(*
 __    __  ______  __    __  ________  __       __   ______   ________  ______   ______    ______  
/  |  /  |/      |/  \  /  |/        |/  \     /  | /      \ /        |/      | /      \  /      \ 
$$ | /$$/ $$$$$$/ $$  \ $$ |$$$$$$$$/ $$  \   /$$ |/$$$$$$  |$$$$$$$$/ $$$$$$/ /$$$$$$  |/$$$$$$  |
$$ |/$$/    $$ |  $$$  \$$ |$$ |__    $$$  \ /$$$ |$$ |__$$ |   $$ |     $$ |  $$ |  $$/ $$ \__$$/ 
$$  $$<     $$ |  $$$$  $$ |$$    |   $$$$  /$$$$ |$$    $$ |   $$ |     $$ |  $$ |      $$      \ 
$$$$$  \    $$ |  $$ $$ $$ |$$$$$/    $$ $$ $$/$$ |$$$$$$$$ |   $$ |     $$ |  $$ |   __  $$$$$$  |
$$ |$$  \  _$$ |_ $$ |$$$$ |$$ |_____ $$ |$$$/ $$ |$$ |  $$ |   $$ |    _$$ |_ $$ \__/  |/  \__$$ |
$$ | $$  |/ $$   |$$ | $$$ |$$       |$$ | $/  $$ |$$ |  $$ |   $$ |   / $$   |$$    $$/ $$    $$/ 
$$/   $$/ $$$$$$/ $$/   $$/ $$$$$$$$/ $$/      $$/ $$/   $$/    $$/    $$$$$$/  $$$$$$/   $$$$$$/  
                                                                                                   
*)

actCheckPositionDeviation();
actCheckRealSpgStatus();
actUpdateDefaults();
actClearDefaults();

startupDelayTON(PT:=T#200MS);
stateDelayTimer(PT:=T#200MS);
timeoutDelay(PT:=T#2S);

actKinematicSetpoints();
actCheckNotMoving();

GVL_INTER.TARGET_MEASUREMENT_ANGLE:= astAxes[AXIS_MEASUREMENT_ANGLE].Axis.NcToPlc.SetPos + astAxes[AXIS_MEASUREMENT_ANGLE_OFFSET].Axis.NcToPlc.SetPos + astAxes[AXIS_ROTATION_SAMPLE].Axis.NcToPlc.SetPos;


FOR i:=1 TO ARRAYSIZE_ALLVIRTUALS DO
    aVirtualAxisDefaults[i].mcSetPosition(Axis:= astAxes[aVirtualAxisDefaults[i].axisID].Axis);
    aVirtualAxisDefaults[i].mcSetPosition.Execute:= FALSE;
END_FOR

IF GVL_INTER.START_RECOVERY AND GVL_INTER.RUN_KINEMATICS AND NOT GVL_INTER.RECOVERY_IN_PROGRESS THEN
    eStateInter:= eState_INTER.startRecovery;
END_IF

IF GVL_INTER.REINITIALISE_IN_PROGRESS THEN
    GVL_INTER.REINITIALISE:= FALSE;
    GVL_INTER.START_RECOVERY:= FALSE;
END_IF
IF GVL_INTER.REINITIALISE_IN_PROGRESS AND eStateInter= eState_INTER.error THEN
    GVL_INTER.REINITIALISE_IN_PROGRESS:= FALSE;
END_IF

IF GVL_INTER.RUN_KINEMATICS AND GVL_INTER.REINITIALISE THEN
    GVL_INTER.RESET_ALL:= TRUE;
    GVL_INTER.REINITIALISE := FALSE;
    GVL_INTER.REINITIALISE_IN_PROGRESS:= TRUE;
    GVL_INTER.RUN_KINEMATICS := FALSE;
END_IF
IF GVL_INTER.FINISH_REINITIALISE AND NOT GVL_INTER.REINITIALISE_IN_PROGRESS THEN
    GVL_INTER.FINISH_REINITIALISE:= FALSE;
END_IF
IF GVL_INTER.FINISH_REINITIALISE AND GVL_INTER.REINITIALISE_IN_PROGRESS THEN
    GVL_INTER.FINISH_REINITIALISE:= FALSE;
    GVL_INTER.RUN_KINEMATICS:= TRUE;
    GVL_INTER.REINITIALISE_IN_PROGRESS:= FALSE;
    eStateInter:= eState_INTER.alignKinematics;
END_IF

IF NOT GVL_INTER.KINEMATIC_SPG_ALL_DISABLED AND NOT GVL_INTER.RUN_KINEMATICS THEN
    eStateInter:= eState_INTER.disableSPG;
END_IF


GVL_INTER.OPERATIONAL:= FALSE;  //OVERRIDE IF OPERATIONAL
IF NOT CombinedVerticalSetupComplete AND GVL_INTER.OPERATIONAL THEN
    eStateInter:= eState_INTER.init;
END_IF
checkRotationDrive(Axis:=astAxes[AXIS_ROTATION].Axis,Enable:=TRUE);

//Sometimes the rotation loads in 360degrees out of phase, we need to be able to detect and fix this.
setPosRotation(Axis:= astAxes[AXIS_ROTATION].Axis, Execute:= FALSE);

IF checkRotationDrive.Valid THEN
    IF ABS(astAxes[AXIS_ROTATION].Axis.NcToPlc.ActPos)>20 AND astAxes[AXIS_ROTATION].Axis.Status.NotMoving THEN
    astAxes[AXIS_ROTATION].stControl.bEnable:= FALSE;
    IF astAxes[AXIS_ROTATION].Axis.NcToPlc.ActPos>20 THEN
        //we need to minus 360
        setPosRotation.Position:= astAxes[AXIS_ROTATION].Axis.NcToPlc.ActPos-360;
    ELSIF astAxes[AXIS_ROTATION].Axis.NcToPlc.ActPos<20 THEN
        //we need to add 360
        setPosRotation.Position:= astAxes[AXIS_ROTATION].Axis.NcToPlc.ActPos+360;
    END_IF
    setPosRotation(Axis:= astAxes[AXIS_ROTATION].Axis, Execute:= TRUE);
ELSE
    bRotationValid:= TRUE;
END_IF
END_IF


IF NOT GVL_INTER.BRAKE_TEST_PASSED THEN
    GVL_INTER.RUN_KINEMATICS := FALSE;
END_IF    
    CASE eStateInter OF
        eState_INTER.init:       
            IF GVL_INTER.RUN_KINEMATICS AND CombinedVerticalSetupComplete AND bRotationValid THEN
                IF GVL_INTER.NC_AXIS_ERROR THEN
                    GVL_INTER.RESET_ALL := TRUE;
                    stateDelayTimer.IN:= TRUE;
                ELSIF NOT stateDelayTimer.IN THEN
                    IF NOT GVL_INTER.KINEMATIC_SPG_ALL_DISABLED THEN
                        eStateInter:=eState_INTER.disableSPG;
                    ELSE
                        IF bRealDevValid THEN
                            eStateInter:= eState_INTER.checkAlignKinematics;
                        ELSE
                            eStateInter:= eState_INTER.setPositions;
						END_IF
                        
			        END_IF
				END_IF
                //To prevent instantaneous reset and no error present
                IF stateDelayTimer.Q THEN
                    stateDelayTimer.IN:= FALSE;
				END_IF
                
			END_IF
            
                        
        eState_INTER.setPositions:
            FOR i:=1 TO ARRAYSIZE_ALLVIRTUALS DO
                aVirtualAxisDefaults[i].mcSetPosition.Position:= aVirtualAxisDefaults[i].defaultPosition ;
                aVirtualAxisDefaults[i].mcSetPosition.Execute:= TRUE;
            END_FOR            
            writeDefault.START:=TRUE;            
            stateDelayTimer.IN:= TRUE;
            IF(stateDelayTimer.Q) THEN
                eStateInter := eState_INTER.checkSetPositions;
                stateDelayTimer.IN:= FALSE;
			END_IF
            
        
        eState_INTER.checkSetPositions:
            IF bDefaultDevValid THEN
                retryCounter:= 0;
                IF bRealDevValid THEN
                    eStateInter:= eState_INTER.enableSPG;
                ELSE
                    eStateInter:= eState_INTER.alignKinematics;
			    END_IF
            ELSE
                IF retryCounter >3 THEN
                    retryCounter:= 0;
                    eStateInter:= eState_INTER.error;
                    GVL_INTER.LOGIC_STATE_ERROR:= eState_INTER.checkSetPositions;
                    GVL_INTER.LOGIC_ERROR:= TRUE;
                ELSE
                    retryCounter:= retryCounter+1;
                    eStateInter:= eState_INTER.setPositions;
				END_IF                
			END_IF               


        eState_INTER.alignKinematics:
            startupDelayTON.IN:= TRUE;
            IF startupDelayTON.Q THEN
                startupDelayTON.IN:= FALSE;
                AbsoluteMove(axisID:= AXIS_HORIZONTAL_TRANSLATION, fPosition:= GVL_INTER.SETPOS_HORIZONTAL);
                AbsoluteMove(axisID:= AXIS_COMBINED_VERTICAL, fPosition:= GVL_INTER.SETPOS_COMBINED_VERTICAL);
                AbsoluteMove(axisID:= AXIS_ROTATION, fPosition:= GVL_INTER.SETPOS_ROTATION);               
                stateDelayTimer.IN:= TRUE;
			END_IF
            IF stateDelayTimer.Q THEN
                eStateInter:= eState_INTER.checkAlignKinematics;
                stateDelayTimer.IN:= FALSE;
			END_IF
            IF NOT (startupDelayTON.IN OR stateDelayTimer.IN) THEN
                GVL_INTER.LOGIC_STATE_ERROR:= eState_INTER.alignKinematics;
                GVL_INTER.LOGIC_ERROR:= TRUE;
                eStateInter:= eState_INTER.error;
			END_IF
            

        eState_INTER.checkAlignKinematics:
            IF GVL_INTER.REAL_AXES_NOT_MOVING THEN   
                timeoutDelay.IN:= TRUE;            
                IF bRealDevValid THEN
                    timeoutDelay.IN:= FALSE;
                    eStateInter:= eState_INTER.enableSPG;
		        END_IF
                IF GVL_INTER.LIMIT_HIT THEN
                    timeoutDelay.IN:= FALSE;
                    GVL_INTER.LOGIC_STATE_ERROR:= eState_INTER.checkAlignKinematics;
                    GVL_INTER.LOGIC_ERROR:= TRUE;
                    eStateInter:= eState_INTER.error;
				END_IF
                IF timeoutDelay.Q THEN
                    timeoutDelay.IN:= FALSE;
                    GVL_INTER.LOGIC_STATE_ERROR:= eState_INTER.checkAlignKinematics;
                    GVL_INTER.LOGIC_ERROR:= TRUE;
                    eStateInter:= eState_INTER.error;
				END_IF
		    END_IF
                
            
        eState_INTER.enableSPG:
            axisSpg_Vertical.spgEnable.Execute:= TRUE;
            axisSpg_Horizontal.spgEnable.Execute:= TRUE;
            axisSpg_Rot.spgEnable.Execute:= TRUE;
            stateDelayTimer.IN:= TRUE;
            IF stateDelayTimer.Q THEN
                stateDelayTimer.IN:= FALSE;
                eStateInter:= eState_INTER.checkEnableSPG;
			END_IF
            
           
        eState_INTER.checkEnableSPG:
            IF GVL_INTER.KINEMATIC_SPG_ALL_ENABLED THEN
                retryCounter:= 0;
                eStateInter :=eState_INTER.operation;
            ELSE
                IF retryCounter >3 THEN
                    retryCounter:= 0;
                    eStateInter:= eState_INTER.error;
                    GVL_INTER.LOGIC_STATE_ERROR:= eState_INTER.checkEnableSPG;
                    GVL_INTER.LOGIC_ERROR:= TRUE;
                ELSE
                    retryCounter:= retryCounter+1;
                    eStateInter:= eState_INTER.enableSPG;
		        END_IF 
			END_IF
            
        
        eState_INTER.operation:
            GVL_INTER.RECOVERY_IN_PROGRESS:= FALSE;
            bKinematicsOperational:= TRUE;
            IF NOT GVL_INTER.KINEMATIC_SPG_ALL_ENABLED THEN
                eStateInter:= eState_INTER.error;
			END_IF
            IF NOT GVL_INTER.NC_AXIS_ERROR THEN
                GVL_INTER.OPERATIONAL:= TRUE;
            END_IF
            
        eState_INTER.disableSPG:
            axisSpg_Vertical.spgDisable.Execute:= TRUE;
            axisSpg_Horizontal.spgDisable.Execute:= TRUE;
            axisSpg_Rot.spgDisable.Execute:= TRUE;
            stateDelayTimer.IN:= TRUE;
            IF stateDelayTimer.Q THEN
                stateDelayTimer.IN:= FALSE;
                eStateInter:= eState_INTER.checkDisableSPG;
			END_IF
            
        eState_INTER.checkDisableSPG:
            IF GVL_INTER.KINEMATIC_SPG_ALL_DISABLED THEN
                retryCounter:= 0;
                IF GVL_INTER.RECOVERY_IN_PROGRESS THEN
                    eStateInter:= eState_INTER.recoveryDefaultPosition;
                ELSE
                    eStateInter:= eState_INTER.init;
				END_IF
            ELSE
                IF retryCounter >3 THEN
                    retryCounter:= 0;
                    eStateInter:= eState_INTER.error;
                    GVL_INTER.LOGIC_STATE_ERROR:= eState_INTER.checkDisableSPG;
                    GVL_INTER.LOGIC_ERROR:= TRUE;
                ELSE
                    retryCounter:= retryCounter+1;
                    eStateInter:= eState_INTER.disableSPG;
		        END_IF 
			END_IF
            
        eState_INTER.startRecovery:
            GVL_INTER.RECOVERY_IN_PROGRESS := TRUE;
            eStateInter:= eState_INTER.disableSPG;
        
        eState_INTER.recoveryDefaultPosition:
            IF GVL_INTER.NC_AXIS_ERROR THEN
                GVL_INTER.RESET_ALL := TRUE;
            ELSE
                FOR i:=1 TO ARRAYSIZE_ALLVIRTUALS DO
                    aVirtualAxisDefaults[i].mcSetPosition.Position:= aVirtualAxisDefaults[i].defaultPosition;
                    aVirtualAxisDefaults[i].mcSetPosition.Execute:= TRUE;
                    aVirtualAxisDefaults[i].mcSetPosition.Options.ClearPositionLag:= TRUE;
                END_FOR
                
                stateDelayTimer.IN:= TRUE;
                IF stateDelayTimer.Q THEN
                    stateDelayTimer.IN:= FALSE;
                    eStateInter:= eState_INTER.waitForRecovery;
			    END_IF
			END_IF
            
          
        eState_INTER.waitForRecovery:
            IF GVL_INTER.VIRTUAL_AXES_NOT_MOVING THEN                
                timeoutDelay.IN:= TRUE;            
                IF bRecoveryDevValid THEN
                    timeoutDelay.IN:= FALSE;
                    GVL_INTER.START_RECOVERY:= FALSE;                    
                    eStateInter:= eState_INTER.init;                                
			    END_IF
                
                IF timeoutDelay.Q THEN
                    timeoutDelay.IN:= FALSE;
                    GVL_INTER.LOGIC_STATE_ERROR:= eState_INTER.waitForRecovery;
                    GVL_INTER.LOGIC_ERROR:= TRUE;
                    GVL_INTER.START_RECOVERY:= FALSE;
                    GVL_INTER.RECOVERY_IN_PROGRESS:= FALSE;
                    eStateInter:= eState_INTER.error;
				END_IF           
			END_IF
            
            
        eState_INTER.error:
            GVL_INTER.RECOVERY_IN_PROGRESS:= FALSE;
            IF GVL_INTER.RESET_REQUESTED THEN
                eStateInter:= eState_INTER.safetyError;
			END_IF
            IF GVL_INTER.ACKNOWLEDGE_LOGIC_ERROR THEN
                GVL_INTER.ACKNOWLEDGE_LOGIC_ERROR := FALSE;
                GVL_INTER.LOGIC_STATE_ERROR:= eState_INTER.none;
                GVL_INTER.LOGIC_ERROR:= FALSE;
                GVL_INTER.RESET_ALL:= TRUE;
			END_IF
            IF GVL_Safety.LocalMode AND GVL_Safety.LocalMode_Disabled THEN
                eStateInter:= eState_INTER.localModeDisabled;
			END_IF
            IF NOT GVL_INTER.NC_AXIS_ERROR  AND NOT GVL_INTER.LOGIC_ERROR THEN
                eStateInter:= eState_INTER.init;
			END_IF
            
        eState_INTER.localModeDisabled:
            IF NOT GVL_INTER.NC_AXIS_ERROR  AND NOT GVL_INTER.LOGIC_ERROR THEN
                eStateInter:= eState_INTER.init;
			END_IF
            
        eState_INTER.safetyError:
            GVL_INTER.RUN_KINEMATICS:= FALSE;
            IF GVL_INTER.ACKNOWLEDGE_LOGIC_ERROR THEN
                GVL_INTER.ACKNOWLEDGE_LOGIC_ERROR := FALSE;
                GVL_INTER.LOGIC_STATE_ERROR:= eState_INTER.none;
                GVL_INTER.LOGIC_ERROR:= FALSE;
                GVL_INTER.RESET_ALL:= TRUE;
			END_IF
            IF NOT GVL_INTER.NC_AXIS_ERROR  AND NOT GVL_INTER.LOGIC_ERROR THEN
                eStateInter:= eState_INTER.init;
			END_IF
            
	END_CASE
    
    IF GVL_INTER.REINITIALISE_IN_PROGRESS OR GVL_INTER.OPERATIONAL THEN   
        FOR i:=1 TO ARRAYSIZE_ALLVIRTUALS DO
            astAxes[aVirtualAxisDefaults[i].axisID].stControl.bEnable:=TRUE;
            astAxes[aVirtualAxisDefaults[i].axisID].stInputs.bLimitBwd:=TRUE;
            astAxes[aVirtualAxisDefaults[i].axisID].stInputs.bLimitFwd:=TRUE;
		END_FOR
    ELSE
        FOR i:=1 TO ARRAYSIZE_ALLVIRTUALS DO
            astAxes[aVirtualAxisDefaults[i].axisID].stControl.bEnable:=FALSE;
            astAxes[aVirtualAxisDefaults[i].axisID].stInputs.bLimitBwd:=FALSE;
            astAxes[aVirtualAxisDefaults[i].axisID].stInputs.bLimitFwd:=FALSE;
		END_FOR
	END_IF

 
//Call set position functions on virtual axes
FOR i:=1 TO ARRAYSIZE_ALLVIRTUALS DO
    aVirtualAxisDefaults[i].mcSetPosition(Axis:=astAxes[aVirtualAxisDefaults[i].axisID].Axis);
    aVirtualAxisDefaults[i].mcSetPosition.Execute:= FALSE;
END_FOR   

GVL_INTER.LOGIC_STATE_STR := TO_STRING(GVL_INTER.LOGIC_STATE);
GVL_INTER.LOGIC_STATE_ERROR_STR := TO_STRING(GVL_INTER.LOGIC_STATE_ERROR);


MC_ExtSetPointGenFeed(Axis:= astAxes[AXIS_COMBINED_VERTICAL].Axis, 
        Position:= axisSpg_Vertical.position,
        Velocity:= axisSpg_Vertical.velocity,
        Direction:= axisSpg_Vertical.direction, Acceleration:= 0);
MC_ExtSetPointGenFeed(Axis:= astAxes[AXIS_HORIZONTAL_TRANSLATION].Axis, 
        Position:= axisSpg_Horizontal.position,
        Velocity:= axisSpg_Horizontal.velocity,
        Direction:= axisSpg_Horizontal.direction, Acceleration:= 0);
MC_ExtSetPointGenFeed(Axis:= astAxes[AXIS_ROTATION].Axis, 
        Position:= axisSpg_Rot.position,
        Velocity:= axisSpg_Rot.velocity,
        Direction:= axisSpg_Rot.direction, Acceleration:= 0);

axisSpg_Vertical.spgEnable(Axis:=astAxes[axisSpg_Vertical.axisID].Axis);
axisSpg_Vertical.spgDisable(Axis:=astAxes[axisSpg_Vertical.axisID].Axis);
axisSpg_Horizontal.spgEnable(Axis:=astAxes[axisSpg_Horizontal.axisID].Axis);
axisSpg_Horizontal.spgDisable(Axis:=astAxes[axisSpg_Horizontal.axisID].Axis);
axisSpg_Rot.spgEnable(Axis:=astAxes[axisSpg_Rot.axisID].Axis);
axisSpg_Rot.spgDisable(Axis:=astAxes[axisSpg_Rot.axisID].Axis);

axisSpg_Vertical.spgEnable.Execute:= FALSE;
axisSpg_Vertical.spgDisable.Execute:= FALSE;
axisSpg_Horizontal.spgEnable.Execute:= FALSE;
axisSpg_Horizontal.spgDisable.Execute:= FALSE;
axisSpg_Rot.spgEnable.Execute:= FALSE;
axisSpg_Rot.spgDisable.Execute:= FALSE;

GVL_INTER.LOGIC_STATE:= eStateInter;

IF ABS( astAxes[AXIS_VERTICAL_TRANSLATION_Y1].stStatus.fActPosition-astAxes[AXIS_VERTICAL_TRANSLATION_Y2].stStatus.fActPosition)>3 THEN
    astAxes[AXIS_COMBINED_VERTICAL].stControl.bEnable:= FALSE;
END_IF

METHOD AbsoluteMove : BOOL
VAR_INPUT
    axisID : UINT;
    fPosition : LREAL;
    
END_VAR
astAxes[axisID].stControl.eCommand:= E_MotionFunctions.eMoveAbsolute;
astAxes[axisID].stControl.fPosition:= fPosition;
astAxes[axisID].stControl.bExecute:= TRUE;
END_METHOD

ACTION actCheckNotMoving:
GVL_INTER.REAL_AXES_NOT_MOVING:= astAxes[AXIS_HORIZONTAL_TRANSLATION].Axis.Status.NotMoving AND astAxes[AXIS_COMBINED_VERTICAL].Axis.Status.NotMoving AND astAxes[AXIS_ROTATION].Axis.Status.NotMoving;

GVL_INTER.VIRTUAL_AXES_NOT_MOVING:= 
    astAxes[AXIS_DOFF_ANGLED].Axis.Status.NotMoving AND
    astAxes[AXIS_DOFF_PARALLEL].Axis.Status.NotMoving AND
    astAxes[AXIS_DTANK_LENGTH].Axis.Status.NotMoving AND
    astAxes[AXIS_DTANK_PIVOT_TO_WINDOW].Axis.Status.NotMoving AND
    astAxes[AXIS_DRAD].Axis.Status.NotMoving AND
    astAxes[AXIS_MEASUREMENT_ANGLE].Axis.Status.NotMoving AND
    astAxes[AXIS_MEASUREMENT_ANGLE_OFFSET].Axis.Status.NotMoving AND
    astAxes[AXIS_ROTATION_CALIBRATION].Axis.Status.NotMoving AND
    astAxes[AXIS_ROTATION_SAMPLE].Axis.Status.NotMoving AND
    astAxes[AXIS_COMBINED_VERTICAL_CALIBRATION].Axis.Status.NotMoving AND
    astAxes[AXIS_COMBINED_VERTICAL_SAMPLE].Axis.Status.NotMoving AND
    astAxes[AXIS_HORIZONTAL_CALIBRATION].Axis.Status.NotMoving AND
    astAxes[AXIS_HORIZONTAL_SAMPLE].Axis.Status.NotMoving;
END_ACTION

ACTION actCheckPositionDeviation:
posDevHorizontal:=    astAxes[AXIS_HORIZONTAL_TRANSLATION].stStatus.fActPosition - GVL_INTER.SETPOS_HORIZONTAL;
posDevVertical:=    astAxes[AXIS_COMBINED_VERTICAL].stStatus.fActPosition - GVL_INTER.SETPOS_COMBINED_VERTICAL;
posDevRot:=    astAxes[AXIS_ROTATION].stStatus.fActPosition - GVL_INTER.SETPOS_ROTATION;

bRealDevValid := ABS(posDevHorizontal)<DEVIATION_THRESHOLD AND ABS(posDevVertical)<DEVIATION_THRESHOLD AND ABS(posDevRot)<DEVIATION_THRESHOLD;

(*
//Check position deviations of "default" axes
bDefaultDevValid:= TRUE; //we will AND it with the deviations in the loop
FOR i := 1 TO ARRAYSIZE_VIRTUALCAL DO
    bDefaultDevValid:= bDefaultDevValid AND (ABS(astAxes[IDs_VirtualWithCalibrationAxes[i]].stStatus.fActPosition - calibrationValuesArray[i])<DEVIATION_THRESHOLD);
END_FOR


//Check position deviations of remaining virtual axes
bRecoveryDevValid:= bDefaultDevValid; //Use default dev as starting point before iterator
FOR i := 1 TO ARRAYSIZE_VIRTUAL DO
    bRecoveryDevValid:= bRecoveryDevValid AND (ABS(astAxes[IDs_VirtualNoCalibrationAxes[i]].stStatus.fActPosition)<DEVIATION_THRESHOLD);
END_FOR
*)

////
////
////
//THIS IS NEW LOGIC THAT OVERRIDES WHAT'S CURRENTLY HAPPENING, BE CAREFUL
bRecoveryDevValid:= TRUE;
FOR i:=1 TO ARRAYSIZE_ALLVIRTUALS DO
    aVirtualAxisDefaults[i].deviation:= ABS(astAxes[aVirtualAxisDefaults[i].axisID].Axis.NcToPlc.ActPos - aVirtualAxisDefaults[i].defaultPosition);
    bRecoveryDevValid:= bRecoveryDevValid AND (aVirtualAxisDefaults[i].deviation<DEVIATION_THRESHOLD);
END_FOR

bDefaultDevValid := bRecoveryDevValid;

bVirtualsMoving:= FALSE;
FOR i := 1 TO ARRAYSIZE_ALLVIRTUALS DO
    bVirtualsMoving:= bVirtualsMoving OR astAxes[aVirtualAxisDefaults[i].axisID].Axis.Status.Moving;
END_FOR
/////
/////
/////
    
    
//bVirtualsMoving:= FALSE;
//Looking for any virtual axis moving IDs_VirtualNoCalibrationAxes
//FOR i := 1 TO ARRAYSIZE_VIRTUALCAL DO
//    bVirtualsMoving:= bVirtualsMoving OR astAxes[IDs_VirtualWithCalibrationAxes[i]].Axis.Status.Moving;
//END_FOR
//FOR i := 1 TO ARRAYSIZE_VIRTUAL DO
//    bVirtualsMoving:= bVirtualsMoving OR astAxes[IDs_VirtualNoCalibrationAxes[i]].Axis.Status.Moving;
//END_FOR
END_ACTION

ACTION actCheckRealSpgStatus:
GVL_INTER.KINEMATIC_SPG_ALL_ENABLED:= astAxes[AXIS_HORIZONTAL_TRANSLATION].Axis.Status.ExtSetPointGenEnabled AND astAxes[AXIS_COMBINED_VERTICAL].Axis.Status.ExtSetPointGenEnabled AND astAxes[AXIS_ROTATION].Axis.Status.ExtSetPointGenEnabled;
GVL_INTER.KINEMATIC_SPG_ALL_DISABLED:= NOT (astAxes[AXIS_HORIZONTAL_TRANSLATION].Axis.Status.ExtSetPointGenEnabled) AND NOT (astAxes[AXIS_COMBINED_VERTICAL].Axis.Status.ExtSetPointGenEnabled) AND NOT (astAxes[AXIS_ROTATION].Axis.Status.ExtSetPointGenEnabled);
END_ACTION

ACTION actClearDefaults:
IF GVL_INTER.CLEAR_ALL_DEFAULTS THEN
    IF NOT bVirtualsMoving THEN
        GVL_INTER.CLEAR_ALL_DEFAULTS:= FALSE;   
        aVirtualAxisDefaults[1].defaultPosition:= 3000;
        aVirtualAxisDefaults[2].defaultPosition:= 2289.15;
        aVirtualAxisDefaults[3].defaultPosition:= 1648.66;
        aVirtualAxisDefaults[4].defaultPosition:= 0;
        aVirtualAxisDefaults[5].defaultPosition:= 0;
        aVirtualAxisDefaults[6].defaultPosition:= 0;
        aVirtualAxisDefaults[7].defaultPosition:= 0;
        aVirtualAxisDefaults[8].defaultPosition:= 0;
        aVirtualAxisDefaults[9].defaultPosition:= 0;
        aVirtualAxisDefaults[10].defaultPosition:= 0;
        aVirtualAxisDefaults[11].defaultPosition:= 0;
        aVirtualAxisDefaults[12].defaultPosition:= 0;
        aVirtualAxisDefaults[13].defaultPosition:= 0;
	END_IF
END_IF
END_ACTION

ACTION actKinematicSetpoints:
(*GVL_INTER.SETPOS_HORIZONTAL:= astAxes[AXIS_HORIZONTAL_VIRTUAL].Axis.NcToPlc.ActPos + astAxes[AXIS_HORIZONTAL_CALIBRATION].Axis.NcToPlc.ActPos + astAxes[AXIS_HORIZONTAL_SAMPLE].Axis.NcToPlc.ActPos;
GVL_INTER.SETVELO_HORIZONTAL:=astAxes[AXIS_HORIZONTAL_VIRTUAL].Axis.NcToPlc.ActVelo + astAxes[AXIS_HORIZONTAL_CALIBRATION].Axis.NcToPlc.ActVelo + astAxes[AXIS_HORIZONTAL_SAMPLE].Axis.NcToPlc.ActVelo;
GVL_INTER.SETPOS_COMBINED_VERTICAL:= astAxes[AXIS_COMBINED_VERTICAL_VIRTUAL].Axis.NcToPlc.ActPos + astAxes[AXIS_COMBINED_VERTICAL_CALIBRATION].Axis.NcToPlc.ActPos + astAxes[AXIS_COMBINED_VERTICAL_SAMPLE].Axis.NcToPlc.ActPos;
GVL_INTER.SETVELO_COMBINED_VERTICAL:= astAxes[AXIS_COMBINED_VERTICAL_VIRTUAL].Axis.NcToPlc.ActVelo + astAxes[AXIS_COMBINED_VERTICAL_CALIBRATION].Axis.NcToPlc.ActVelo + astAxes[AXIS_COMBINED_VERTICAL_SAMPLE].Axis.NcToPlc.ActVelo;
GVL_INTER.SETPOS_ROTATION:= astAxes[AXIS_ROTATION_VIRTUAL].Axis.NcToPlc.ActPos + astAxes[AXIS_ROTATION_CALIBRATION].Axis.NcToPlc.ActPos + astAxes[AXIS_ROTATION_SAMPLE].Axis.NcToPlc.ActPos;
GVL_INTER.SETVELO_ROTATION:= astAxes[AXIS_ROTATION_VIRTUAL].Axis.NcToPlc.ActVelo + astAxes[AXIS_ROTATION_CALIBRATION].Axis.NcToPlc.ActVelo + astAxes[AXIS_ROTATION_SAMPLE].Axis.NcToPlc.ActVelo;

//Horizontal direction
IF GVL_INTER.SETVELO_HORIZONTAL >0 THEN
    GVL_INTER.SETDIR_HORIZONTAL := 1;
ELSIF GVL_INTER.SETVELO_HORIZONTAL<0 THEN
    GVL_INTER.SETDIR_HORIZONTAL := -1;
ELSE
    GVL_INTER.SETDIR_HORIZONTAL := 0;
END_IF

//Vertical Direction
IF GVL_INTER.SETVELO_COMBINED_VERTICAL>0 THEN
    GVL_INTER.SETDIR_COMBINED_VERTICAL := 1;
ELSIF GVL_INTER.SETVELO_COMBINED_VERTICAL<0 THEN
    GVL_INTER.SETDIR_COMBINED_VERTICAL := -1;
ELSE
    GVL_INTER.SETDIR_COMBINED_VERTICAL := 0;
END_IF

//Rotation direction
IF GVL_INTER.SETVELO_ROTATION>0 THEN
    GVL_INTER.SETDIR_ROTATION := 1;
ELSIF GVL_INTER.SETVELO_ROTATION<0 THEN
    GVL_INTER.SETDIR_ROTATION := -1;
ELSE
    GVL_INTER.SETDIR_ROTATION := 0;
END_IF
*)

//NEW LOGIC
axisSpg_Vertical.position:= astAxes[AXIS_COMBINED_VERTICAL_VIRTUAL].Axis.NcToPlc.ActPos + astAxes[AXIS_COMBINED_VERTICAL_CALIBRATION].Axis.NcToPlc.ActPos + astAxes[AXIS_COMBINED_VERTICAL_SAMPLE].Axis.NcToPlc.ActPos;
axisSpg_Horizontal.position:= astAxes[AXIS_HORIZONTAL_VIRTUAL].Axis.NcToPlc.ActPos + astAxes[AXIS_HORIZONTAL_CALIBRATION].Axis.NcToPlc.ActPos + astAxes[AXIS_HORIZONTAL_SAMPLE].Axis.NcToPlc.ActPos;
//axisSpg_Rot.position:= astAxes[AXIS_ROTATION_VIRTUAL].Axis.NcToPlc.ActPos + astAxes[AXIS_ROTATION_CALIBRATION].Axis.NcToPlc.ActPos + astAxes[AXIS_ROTATION_SAMPLE].Axis.NcToPlc.ActPos;

axisSpg_Rot.position:= astAxes[AXIS_ROTATION_VIRTUAL].Axis.NcToPlc.ActPos + astAxes[AXIS_ROTATION_CALIBRATION].Axis.NcToPlc.ActPos;

axisSpg_Vertical.velocity:= astAxes[AXIS_COMBINED_VERTICAL_VIRTUAL].Axis.NcToPlc.ActVelo + astAxes[AXIS_COMBINED_VERTICAL_CALIBRATION].Axis.NcToPlc.ActVelo + astAxes[AXIS_COMBINED_VERTICAL_SAMPLE].Axis.NcToPlc.ActVelo;
axisSpg_Horizontal.velocity:=astAxes[AXIS_HORIZONTAL_VIRTUAL].Axis.NcToPlc.ActVelo + astAxes[AXIS_HORIZONTAL_CALIBRATION].Axis.NcToPlc.ActVelo + astAxes[AXIS_HORIZONTAL_SAMPLE].Axis.NcToPlc.ActVelo;
//axisSpg_Rot.velocity:= astAxes[AXIS_ROTATION_VIRTUAL].Axis.NcToPlc.ActVelo + astAxes[AXIS_ROTATION_CALIBRATION].Axis.NcToPlc.ActVelo + astAxes[AXIS_ROTATION_SAMPLE].Axis.NcToPlc.ActVelo;
axisSpg_Rot.velocity:= astAxes[AXIS_ROTATION_VIRTUAL].Axis.NcToPlc.ActVelo + astAxes[AXIS_ROTATION_CALIBRATION].Axis.NcToPlc.ActVelo;

//Horizontal direction
IF axisSpg_Horizontal.velocity >0 THEN
    axisSpg_Horizontal.direction := 1;
ELSIF axisSpg_Horizontal.velocity<0 THEN
    axisSpg_Horizontal.direction := -1;
ELSE
    axisSpg_Horizontal.direction := 0;
END_IF

//Vertical direction
IF axisSpg_Vertical.velocity >0 THEN
    axisSpg_Vertical.direction := 1;
ELSIF axisSpg_Vertical.velocity<0 THEN
    axisSpg_Vertical.direction := -1;
ELSE
    axisSpg_Vertical.direction := 0;
END_IF

//Rotation direction
IF axisSpg_Rot.velocity >0 THEN
    axisSpg_Rot.direction := 1;
ELSIF axisSpg_Rot.velocity<0 THEN
    axisSpg_Rot.direction := -1;
ELSE
    axisSpg_Rot.direction := 0;
END_IF


//Transfer values over to GVL_INTER
GVL_INTER.SETPOS_HORIZONTAL:=axisSpg_Horizontal.position;
GVL_INTER.SETVELO_HORIZONTAL:=axisSpg_Horizontal.velocity;
GVL_INTER.SETDIR_HORIZONTAL:= axisSpg_Horizontal.direction;

GVL_INTER.SETPOS_COMBINED_VERTICAL:= axisSpg_Vertical.position;
GVL_INTER.SETVELO_COMBINED_VERTICAL:= axisSpg_Vertical.velocity;
GVL_INTER.SETDIR_COMBINED_VERTICAL:= axisSpg_Vertical.direction;

GVL_INTER.SETPOS_ROTATION:= axisSpg_Rot.position;
GVL_INTER.SETVELO_ROTATION:= axisSpg_Rot.velocity;
GVL_INTER.SETDIR_ROTATION:= axisSpg_Rot.direction;
END_ACTION

ACTION actSafeSpeedSwitching:
IF GVL_Safety.UnoccupiedMode THEN
    //HIGH SPEED
    //MEASUREMENT AXIS valid at 0.65 degs/s  
    //Verts max at 27.5
    //Rot at 0.65
    //Hor at 1.3
    //
    FOR i:=1 TO ARRAYSIZE_ALLVIRTUALS DO
        astAxes[aVirtualAxisDefaults[i].axisID].stConfig.fOverride := 100;
        GVL_INTER.SPEED_LIMITING:= FALSE;
	END_FOR
ELSE
    //LOW SPEED
    FOR i:=1 TO ARRAYSIZE_ALLVIRTUALS DO
        astAxes[aVirtualAxisDefaults[i].axisID].stConfig.fOverride := LOCALMODE_SPEED_OVERRIDE * LOCALMODE_SPEED_OVERRIDE_MODIFIER;
        GVL_INTER.SPEED_LIMITING:= TRUE;
	END_FOR
END_IF



(*
//Check speeds not too high
IF NOT GVL_INTER.SPEED_LIMITING AND (ABS(axisSpg_Vertical.velocity)>VERTICAL_SPEED_LIMIT OR ABS(axisSpg_Horizontal.velocity)>HORIZONTAL_SPEED_LIMIT OR ABS(axisSpg_Rot.velocity)>ROTATION_SPEED_LIMIT) THEN
    IF axisSpg_Vertical.velocity>0 THEN
        axisSpg_Vertical.velocity:= VERTICAL_SPEED_LIMIT;
    ELSE
        axisSpg_Vertical.velocity:= -VERTICAL_SPEED_LIMIT;
    END_IF    
    
    IF axisSpg_Horizontal.velocity>0 THEN
        axisSpg_Horizontal.velocity:= HORIZONTAL_SPEED_LIMIT;
    ELSE
        axisSpg_Horizontal.velocity:= -HORIZONTAL_SPEED_LIMIT;
    END_IF 
    
     IF axisSpg_Rot.velocity>0 THEN
        axisSpg_Rot.velocity:= ROTATION_SPEED_LIMIT;
    ELSE
        axisSpg_Rot.velocity:= -ROTATION_SPEED_LIMIT;
    END_IF 

    FOR i:=1 TO ARRAYSIZE_ALLVIRTUALS DO
        astAxes[aVirtualAxisDefaults[i].axisID].stConfig.fOverride := 20;
        GVL_INTER.SPEED_LIMITING:= TRUE;
	END_FOR
END_IF
//We have stopped moving so can stop speed limiting
IF GVL_INTER.VIRTUAL_AXES_NOT_MOVING AND GVL_INTER.SPEED_LIMITING THEN
    FOR i:=1 TO ARRAYSIZE_ALLVIRTUALS DO
        astAxes[aVirtualAxisDefaults[i].axisID].stConfig.fOverride := 100;
        GVL_INTER.SPEED_LIMITING:= FALSE;
	END_FOR
END_IF
*)
END_ACTION

ACTION actSyncVertStateMachine:
CombinedVerticalSetupComplete := FALSE;
vertTon(PT:=T#100MS);
vertDelay(PT:=T#100MS);
CASE eStateVertical OF
        eState_Vertical.init:
            IF NOT astAxes[AXIS_VERTICAL_TRANSLATION_Y1].Axis.STatus.Error OR NOT astAxes[AXIS_VERTICAL_TRANSLATION_Y2].Axis.Status.Error THEN
                IF NOT GVL_INTER.DECOUPLE_VERTICAL_AXES THEN
                    eStateVertical := eState_Vertical.checkPosition;
                END_IF
			END_IF
            
        eState_Vertical.checkPosition:
            vertDelay.IN:= TRUE;
            IF ABS(astAxes[AXIS_VERTICAL_TRANSLATION_Y1].stStatus.fActPosition - astAxes[AXIS_VERTICAL_TRANSLATION_Y2].stStatus.fActPosition)>0.02 THEN
                AbsoluteMove(axisID:=AXIS_VERTICAL_TRANSLATION_Y2,fPosition:= astAxes[AXIS_VERTICAL_TRANSLATION_Y1].stStatus.fActPosition);
			    bVertCorrectionInProgress:= TRUE;
            END_IF
            IF vertDelay.Q AND astAxes[AXIS_VERTICAL_TRANSLATION_Y2].Axis.Status.NotMoving THEN
                bVertCorrectionInProgress:= FALSE;
			END_IF
            IF NOT bVertCorrectionInProgress THEN
                vertDelay.IN:= FALSE;
                eStateVertical := eState_Vertical.setPosition; //should be setPosition state
			END_IF
            
            //Assume Z1 and Z2 calibrated to be at same position
            //IF ABS(fVerticalSimulatedDeviation)> fVerticalSimulatedDeviationAllowed THEN
            //ELSE
                //eStateVertical := eState_Vertical.enableSpg;
			//END_IF
            
        eState_Vertical.setPosition:
            combinedVerticalSetPos.Position:= astAxes[AXIS_VERTICAL_TRANSLATION_Y1].stStatus.fActPosition;
            combinedVerticalSetPos.Execute:= TRUE;
            //eStateVertical := eState_Vertical.checkPosition;
            vertTon.In := TRUE;
            IF vertTon.Q THEN
                eStateVertical := eState_Vertical.enableSpg;
                vertTon.IN:= FALSE;
			END_IF
            
            
        eState_Vertical.enableSpg:
        
            IF astAxes[AXIS_COMBINED_VERTICAL].stInputs.bLimitBwd AND astAxes[AXIS_COMBINED_VERTICAL].stInputs.bLimitFwd THEN
                verticalZ1SpgEnable.Execute := TRUE;
                verticalZ2SpgEnable.Execute := TRUE;
                eStateVertical := eState_Vertical.confirmEnableSpg;
            ELSE
                tempZ1Power(Axis:= astAxes[AXIS_VERTICAL_TRANSLATION_Y1].Axis, Enable:= TRUE, Enable_Negative:=TRUE, Enable_Positive:=TRUE);
			    tempZ2Power(Axis:= astAxes[AXIS_VERTICAL_TRANSLATION_Y2].Axis, Enable:= TRUE, Enable_Negative:=TRUE, Enable_Positive:=TRUE);
                verticalZ1SpgEnable.Execute := TRUE;
                verticalZ2SpgEnable.Execute := TRUE;
                eStateVertical := eState_Vertical.confirmEnableSpg;
            END_IF
            
        
        eState_Vertical.confirmEnableSpg:
            confirmSpgTimeout.IN:= TRUE;
            //Timeout check
            IF confirmSpgTimeout.Q THEN
                confirmSpgTimeout.IN:= FALSE;
                eStateVertical := eState_Vertical.init;
			END_IF
            IF VerticalAxesSpgEnabled THEN
                eStateVertical := eState_Vertical.operation;
			END_IF
        
        eState_Vertical.operation:
            //DO NOTHING
            CombinedVerticalSetupComplete := TRUE;
            IF NOT VerticalAxesSpgEnabled THEN
                eStateVertical:= eState_Vertical.init;
			END_IF
            IF astAxes[AXIS_VERTICAL_TRANSLATION_Y1].Axis.STatus.Error OR astAxes[AXIS_VERTICAL_TRANSLATION_Y2].Axis.Status.Error THEN
                eStateVertical:= eState_Vertical.init;
			END_IF
            IF GVL_INTER.DECOUPLE_VERTICAL_AXES THEN
                eStateVertical := eState_Vertical.disableSpg;
			END_IF
            (*IF astAxes[AXIS_COMBINED_VERTICAL].Axis.Status.NotMoving THEN
                IF ABS(astAxes[AXIS_COMBINED_VERTICAL].stStatus.fActPosition-astAxes[AXIS_VERTICAL_TRANSLATION_Y1].stStatus.fActPosition)>0.02 THEN
                    combinedVerticalSetPos.Position:= astAxes[AXIS_VERTICAL_TRANSLATION_Y1].stStatus.fActPosition;
                    combinedVerticalSetPos.Execute:= TRUE;
				END_IF
			END_IF*)
            
        eState_Vertical.disableSpg:
            verticalZ1SpgDisable.Execute:= TRUE;
            verticalZ2SpgDisable.Execute:= TRUE;
            eStateVertical := eState_Vertical.confirmDisableSpg;
            
        eState_Vertical.confirmDisableSpg:
            IF NOT astAxes[AXIS_VERTICAL_TRANSLATION_Y1].Axis.Status.ExtSetPointGenEnabled AND NOT astAxes[AXIS_VERTICAL_TRANSLATION_Y2].Axis.Status.ExtSetPointGenEnabled THEN
                eStateVertical := eState_Vertical.init;
            ELSE
                eStateVertical := eState_Vertical.disableSpg;
			END_IF
            
	END_CASE
END_ACTION

ACTION actUpdateDefaults:
IF GVL_INTER.UPDATE_DEFAULTS THEN
    IF NOT bVirtualsMoving THEN
        GVL_INTER.UPDATE_DEFAULTS:= FALSE;   
        FOR i:=1 TO ARRAYSIZE_ALLVIRTUALS DO
            aVirtualAxisDefaults[i].defaultPosition:= astAxes[aVirtualAxisDefaults[i].axisID].Axis.NcToPlc.ActPos;
        END_FOR
	END_IF
END_IF
END_ACTION

ACTION actZSetpoints:
astAxes[AXIS_COMBINED_VERTICAL].Axis.ReadStatus();
astAxes[AXIS_VERTICAL_TRANSLATION_Y1].Axis.ReadStatus();
astAxes[AXIS_VERTICAL_TRANSLATION_Y2].Axis.ReadStatus();

fY1_To_Simulated_Deviation := astAxes[AXIS_COMBINED_VERTICAL].Axis.NcToPlc.SetPos - astAxes[AXIS_VERTICAL_TRANSLATION_Y1].Axis.NcToPlc.ActPos;
fY2_To_Simulated_Deviation := astAxes[AXIS_COMBINED_VERTICAL].Axis.NcToPlc.SetPos - astAxes[AXIS_VERTICAL_TRANSLATION_Y2].Axis.NcToPlc.ActPos;
/////////////////////


//No move previously in progress
IF ABS(fY2_To_Simulated_Deviation) > 0.01 AND astAxes[AXIS_COMBINED_VERTICAL].Axis.Status.NotMoving AND y2NotFinished=FALSE THEN
    y2Compensating:= TRUE;
    y2NotFinished:= TRUE;
    y2CompensatingCycle:=0;
    //Latch the deviation
    fY2_To_Simulated_Deviation_Latched:= fY2_To_Simulated_Deviation;
ELSIF astAxes[AXIS_COMBINED_VERTICAL].Axis.Status.Moving THEN
    y2NotFinished:= TRUE;
END_IF
//We are compensating and moving forward
IF y2Compensating THEN
    
    IF astAxes[AXIS_COMBINED_VERTICAL].Axis.NcToPlc.ActVelo >0  THEN
        //Moving forward and REAL is LAGGING!!!
        IF fY2_To_Simulated_Deviation_Latched>0 THEN
            fZ2SetPos:= astAxes[AXIS_COMBINED_VERTICAL].Axis.NcToPlc.SetPos - fY2_To_Simulated_Deviation_Latched + ((fY2_To_Simulated_Deviation_Latched/CYCLES_TO_COMPENSATE)*y2CompensatingCycle);
            y2CompensatingCycle:= y2CompensatingCycle+1;
            fZ2SetVelo:=astAxes[AXIS_COMBINED_VERTICAL].Axis.NcToPlc.SetVelo;
            imHere:=7;
        //Moving forward and REAL is LEADING!!!
        ELSIF fY2_To_Simulated_Deviation_Latched<0 THEN
            fZ2SetPos:= astAxes[AXIS_COMBINED_VERTICAL].Axis.NcToPlc.SetPos - fY2_To_Simulated_Deviation_Latched + ((fY2_To_Simulated_Deviation_Latched/CYCLES_TO_COMPENSATE)*y2CompensatingCycle);
            y2CompensatingCycle:= y2CompensatingCycle+1;
            fZ2SetVelo:=astAxes[AXIS_COMBINED_VERTICAL].Axis.NcToPlc.SetVelo;

		END_IF
    ELSIF astAxes[AXIS_COMBINED_VERTICAL].Axis.NcToPlc.ActVelo <0 THEN
        //Moving backward and REAL is LAGGING!!!
        IF fY2_To_Simulated_Deviation_Latched<0 THEN
            fZ2SetPos:= astAxes[AXIS_COMBINED_VERTICAL].Axis.NcToPlc.SetPos - fY2_To_Simulated_Deviation_Latched + ((fY2_To_Simulated_Deviation_Latched/CYCLES_TO_COMPENSATE)*y2CompensatingCycle);
            y2CompensatingCycle:= y2CompensatingCycle+1;
            fZ2SetVelo:=astAxes[AXIS_COMBINED_VERTICAL].Axis.NcToPlc.SetVelo;
            imHere:=4;
        //Moving backward and REAL is LEADING!!!
        ELSIF fY2_To_Simulated_Deviation_Latched>0 THEN
            fZ2SetPos:= astAxes[AXIS_COMBINED_VERTICAL].Axis.NcToPlc.SetPos - fY2_To_Simulated_Deviation_Latched + ((fY2_To_Simulated_Deviation_Latched/CYCLES_TO_COMPENSATE)*y2CompensatingCycle);
            y2CompensatingCycle:= y2CompensatingCycle+1;
            fZ2SetVelo:=astAxes[AXIS_COMBINED_VERTICAL].Axis.NcToPlc.SetVelo;

		END_IF
	END_IF
    
ELSE
   imHere:=1;
  fZ2SetVelo:=astAxes[AXIS_COMBINED_VERTICAL].Axis.NcToPlc.SetVelo;
  fZ2SetPos:= astAxes[AXIS_COMBINED_VERTICAL].Axis.NcToPlc.SetPos;
END_IF
IF y2CompensatingCycle>CYCLES_TO_COMPENSATE THEN
    y2Compensating:= FALSE;
    y2CompensatingCycle:=0;
END_IF
/////////////////////////////////////
////////////////
IF ABS(fY1_To_Simulated_Deviation) > 0.01 AND astAxes[AXIS_COMBINED_VERTICAL].Axis.Status.NotMoving AND y1NotFinished=FALSE THEN
    y1Compensating:= TRUE;
    y1NotFinished:= TRUE;
    y1CompensatingCycle:=0;
    //Latch the deviation
    fY1_To_Simulated_Deviation_Latched:= fY1_To_Simulated_Deviation;
ELSIF astAxes[AXIS_COMBINED_VERTICAL].Axis.Status.Moving THEN
    y1NotFinished:= TRUE;
END_IF
//We are compensating and moving forward
IF y1Compensating THEN
    
    IF astAxes[AXIS_COMBINED_VERTICAL].Axis.NcToPlc.ActVelo >0  THEN
        //Moving forward and REAL is LAGGING!!!
        IF fY1_To_Simulated_Deviation_Latched>0 THEN
            fZ1SetPos:= astAxes[AXIS_COMBINED_VERTICAL].Axis.NcToPlc.SetPos - fY1_To_Simulated_Deviation_Latched + ((fY1_To_Simulated_Deviation_Latched/CYCLES_TO_COMPENSATE)*y1CompensatingCycle);
            y1CompensatingCycle:= y1CompensatingCycle+1;
            fZ1SetVelo:=astAxes[AXIS_COMBINED_VERTICAL].Axis.NcToPlc.SetVelo;
            imHere:=7;
        //Moving forward and REAL is LEADING!!!
        ELSIF fY1_To_Simulated_Deviation_Latched<0 THEN
            fZ1SetPos:= astAxes[AXIS_COMBINED_VERTICAL].Axis.NcToPlc.SetPos - fY1_To_Simulated_Deviation_Latched + ((fY1_To_Simulated_Deviation_Latched/CYCLES_TO_COMPENSATE)*y1CompensatingCycle);
            y1CompensatingCycle:= y1CompensatingCycle+1;
            fZ1SetVelo:=astAxes[AXIS_COMBINED_VERTICAL].Axis.NcToPlc.SetVelo;
		END_IF
    ELSIF astAxes[AXIS_COMBINED_VERTICAL].Axis.NcToPlc.ActVelo <0 THEN
        //Moving backward and REAL is LAGGING!!!
        IF fY1_To_Simulated_Deviation_Latched<0 THEN
            fZ1SetPos:= astAxes[AXIS_COMBINED_VERTICAL].Axis.NcToPlc.SetPos - fY1_To_Simulated_Deviation_Latched + ((fY1_To_Simulated_Deviation_Latched/CYCLES_TO_COMPENSATE)*y1CompensatingCycle);
            y1CompensatingCycle:= y1CompensatingCycle+1;
            fZ1SetVelo:=astAxes[AXIS_COMBINED_VERTICAL].Axis.NcToPlc.SetVelo;
            imHere:=4;
        //Moving backward and REAL is LEADING!!!
        ELSIF fY1_To_Simulated_Deviation_Latched>0 THEN
            fZ1SetPos:= astAxes[AXIS_COMBINED_VERTICAL].Axis.NcToPlc.SetPos - fY1_To_Simulated_Deviation_Latched + ((fY1_To_Simulated_Deviation_Latched/CYCLES_TO_COMPENSATE)*y1CompensatingCycle);
            y1CompensatingCycle:= y1CompensatingCycle+1;
            fZ1SetVelo:=astAxes[AXIS_COMBINED_VERTICAL].Axis.NcToPlc.SetVelo;

		END_IF
	END_IF
    
ELSE
   imHere:=1;
  fZ1SetVelo:=astAxes[AXIS_COMBINED_VERTICAL].Axis.NcToPlc.SetVelo;
  fZ1SetPos:= astAxes[AXIS_COMBINED_VERTICAL].Axis.NcToPlc.SetPos;

END_IF
IF y1CompensatingCycle>CYCLES_TO_COMPENSATE THEN
    y1Compensating:= FALSE;
    y1CompensatingCycle:=0;
END_IF



////////////
////////////////////////
IF astAxes[AXIS_COMBINED_VERTICAL].Axis.NcToPlc.ActVelo =0 THEN
    y2NotFinished:= FALSE;
    y2Compensating:= FALSE;
    y2CompensatingCycle:=0;
    y1NotFinished:= FALSE;
    y1Compensating:= FALSE;
    y1CompensatingCycle:=0;
END_IF
(*
IF combinedVerticalDirection=0 THEN
    y2NotFinished:= FALSE;
    y1NotFinished:= FALSE;
    y2Compensating:= FALSE;
    y2CompensatingCycle:=0;
    y1Compensating:= FALSE;
    y1CompensatingCycle:=0;
END_IF*)
///////////////////////////////////
//OVERRIDE
//fZ1SetPos:= astAxes[AXIS_COMBINED_VERTICAL].Axis.NcToPlc.SetPos;
//fZ1SetVelo :=astAxes[AXIS_COMBINED_VERTICAL].Axis.NcToPlc.SetVelo;



//fZ1SetPos := astAxes[AXIS_COMBINED_VERTICAL].Axis.NcToPlc.SetPos; // DON'T MOVE
//fZ1SetVelo :=astAxes[AXIS_COMBINED_VERTICAL].Axis.NcToPlc.SetVelo;
fZ1SetDir := combinedVerticalDirection;

//fZ2SetPos := astAxes[AXIS_COMBINED_VERTICAL].Axis.NcToPlc.SetPos; // DON'T MOVE
fZ2SetDir := combinedVerticalDirection;
    
MC_ExtSetPointGenFeed(Axis:=astAxes[AXIS_VERTICAL_TRANSLATION_Y1].Axis, Position:= fZ1SetPos, Velocity:= fZ1SetVelo, Acceleration:= 0, Direction:= fZ1SetDir);
MC_ExtSetPointGenFeed(Axis:=astAxes[AXIS_VERTICAL_TRANSLATION_Y2].Axis, Position:= fZ2SetPos, Velocity:= fZ2SetVelo, Acceleration:= 0, Direction:= fZ2SetDir);
END_ACTION

METHOD CheckNcErrors : BOOL
VAR_INPUT
END_VAR
VAR
    i : UINT := 5;
    Error : BOOL := FALSE;
END_VAR
FOR i :=5 TO GVL_APP.nAXIS_NUM DO
    IF astAxes[i].stStatus.bError THEN
        Error := TRUE;
	END_IF
END_FOR
CheckNcErrors := Error;
END_METHOD

METHOD CheckRealLimits : BOOL
VAR_INPUT
END_VAR
//TRUE ON LIMIT HIT
CheckRealLimits:= NOT(astAxes[AXIS_ROTATION].stInputs.bLimitBwd) OR NOT(astAxes[AXIS_ROTATION].stInputs.bLimitFwd) OR
    NOT(astAxes[AXIS_COMBINED_VERTICAL].stInputs.bLimitBwd) OR NOT(astAxes[AXIS_COMBINED_VERTICAL].stInputs.bLimitFwd) OR
    NOT(astAxes[AXIS_HORIZONTAL_TRANSLATION].stInputs.bLimitBwd) OR NOT(astAxes[AXIS_HORIZONTAL_TRANSLATION].stInputs.bLimitFwd);
END_METHOD

METHOD CheckVerticalCalibration : BOOL
VAR_INPUT
END_VAR
CheckVerticalCalibration := astAxes[AXIS_VERTICAL_TRANSLATION_Y2].Axis.Status.Homed AND astAxes[AXIS_VERTICAL_TRANSLATION_Y1].Axis.Status.Homed;
END_METHOD

METHOD CheckZSpgStatus : BOOL
VAR
    SpgSet : BOOL := FALSE;
END_VAR
SpgSet := astAxes[AXIS_VERTICAL_TRANSLATION_Y1].Axis.Status.ExtSetPointGenEnabled AND astAxes[AXIS_VERTICAL_TRANSLATION_Y2].Axis.Status.ExtSetPointGenEnabled;
CheckZSpgStatus := SpgSet;
END_METHOD

METHOD DisableAxes : BOOL
VAR_INPUT
END_VAR
astAxes[AXIS_HORIZONTAL_TRANSLATION].stControl.bEnable :=FALSE;
astAxes[AXIS_VERTICAL_TRANSLATION_Y2].stControl.bEnable :=FALSE;
astAxes[AXIS_VERTICAL_TRANSLATION_Y1].stControl.bEnable :=FALSE;
astAxes[AXIS_ROTATION].stControl.bEnable :=FALSE;
GVL_INTER.DISABLE_ALL_AXES := FALSE;
END_METHOD

METHOD EnableAxes : BOOL
VAR_INPUT
END_VAR
astAxes[AXIS_HORIZONTAL_TRANSLATION].stControl.bEnable :=TRUE;
astAxes[AXIS_VERTICAL_TRANSLATION_Y2].stControl.bEnable :=TRUE;
astAxes[AXIS_VERTICAL_TRANSLATION_Y1].stControl.bEnable :=TRUE;
astAxes[AXIS_ROTATION].stControl.bEnable :=TRUE;
GVL_INTER.ENABLE_ALL_AXES := FALSE;
END_METHOD

METHOD ResetAll : BOOL
VAR_INPUT
END_VAR

VAR
    i : UINT :=5;
END_VAR
FOR i :=1 TO GVL_APP.nAXIS_NUM DO
    IF astAxes[i].stStatus.bError OR astAxes[i].Axis.Status.Error THEN
        astAxes[i].stControl.bReset:= TRUE;
	END_IF      
END_FOR

GVL_INTER.RESET_ALL := FALSE;
END_METHOD

END_PROGRAM

// ---- POUs/Application_Specific/Applications/VirtualSpeedOverrides.TcPOU
PROGRAM VirtualSpeedOverrides
VAR
    i : INT :=0; //iterator for FOR loops
    
    LOCALMODE_SPEED_OVERRIDE : LREAL := 18; //Local mode override of base 20%
    SPEED_OVERRIDE_MODIFIER : LREAL := 1; //Proportional modifier to local mode speed
    
    VerticalOverride : LREAL := 1;
    HorizontalOverride : LREAL := 1;
    RotationOverride : LREAL := 1;
    
    bTest : BOOL;
    
END_VAR
VAR CONSTANT
    VERTICAL_MECHANICAL_LIMIT : LREAL := 28;
    HORIZONTAL_MECHANICAL_LIMIT : LREAL := 5; //Not actually but just no need to be fast
    ROTATION_MECHANICAL_LIMIT : LREAL := 0.65; // Not actually, just a sensible number
    
    VERTICAL_SAFE_LIMIT : LREAL := 5;
    HORIZONTAL_SAFE_LIMIT : LREAL := 5;
    ROTATION_SAFE_LIMIT : LREAL := 0.15;
    
    
    
    THRESHOLD : LREAL := 0.8; //May need to tune this, this'll be the limit we start overriding at so we don't trip the actual mechanical or safe limits
    NON_LINEAR_FUDGE_FACTOR :LREAL := 0.75;
END_VAR

(*Latest thoughts,
K.I.S.S

Look at the setpoint velocities of each real axis
Work out which axis is suffering worse
We can back calculate the original setpoint by dividing throuhgh the override value
We constantly back calculate so we can change the override every cycle

I think we keep the flat local mode speed override - should stop any instantaneous overspeeds I can't catch
But we'll monitor for 80%? within mechanical and safe limits
*)

IF GVL_Safety.UnoccupiedMode THEN   
    //Check vertical axis
    IF (ABS(INTER_LOGIC.axisSpg_Vertical.velocity)) > (VERTICAL_MECHANICAL_LIMIT*THRESHOLD) THEN
        VerticalOverride:= ((VERTICAL_MECHANICAL_LIMIT*THRESHOLD)/ABS(INTER_LOGIC.axisSpg_Vertical.velocity))*NON_LINEAR_FUDGE_FACTOR;
    ELSE
        VerticalOverride:= 1;//No vertical limiting required
	END_IF
    
    //Check horizontal axis
    IF (ABS(INTER_LOGIC.axisSpg_Horizontal.velocity)) > (HORIZONTAL_MECHANICAL_LIMIT*THRESHOLD) THEN
        HorizontalOverride:= ((HORIZONTAL_MECHANICAL_LIMIT*THRESHOLD)/ABS(INTER_LOGIC.axisSpg_Horizontal.velocity))*NON_LINEAR_FUDGE_FACTOR;
    ELSE
        HorizontalOverride:= 1;//No horizontal limiting required
	END_IF
    
    //Check rotation axis
    IF (ABS(INTER_LOGIC.axisSpg_Rot.velocity)) > (ROTATION_MECHANICAL_LIMIT*THRESHOLD) THEN
        RotationOverride:= (ROTATION_MECHANICAL_LIMIT*THRESHOLD)/ABS(INTER_LOGIC.axisSpg_Rot.velocity);
    ELSE
        RotationOverride:= 1;//No rotation limiting required
	END_IF
        
    SPEED_OVERRIDE_MODIFIER:= MIN(VerticalOverride, HorizontalOverride, RotationOverride);  //Take the worst case scenario
    
    FOR i:=1 TO INTER_LOGIC.ARRAYSIZE_ALLVIRTUALS DO
        astAxes[INTER_LOGIC.aVirtualAxisDefaults[i].axisID].stConfig.fOverride := 100* SPEED_OVERRIDE_MODIFIER;
        
	END_FOR
    FOR i:=1 TO 3 DO
        astAxes[AXIS_COMBINED_VERTICAL].stConfig.fOverride := 100;
        astAxes[AXIS_ROTATION].stConfig.fOverride := 100;
        astAxes[AXIS_HORIZONTAL_TRANSLATION].stConfig.fOverride := 100;
	END_FOR

ELSE
    //LOW SPEED MODE
    FOR i:=1 TO 3 DO
        astAxes[AXIS_COMBINED_VERTICAL].stConfig.fOverride := LOCALMODE_SPEED_OVERRIDE;
        astAxes[AXIS_ROTATION].stConfig.fOverride :=LOCALMODE_SPEED_OVERRIDE;
        astAxes[AXIS_HORIZONTAL_TRANSLATION].stConfig.fOverride := LOCALMODE_SPEED_OVERRIDE;
	END_FOR
    //Unsure on this maths, the spgs are created from the axes that will have by default had a 20% speed override applied, so I don't need to use that in initial caluclation?
    IF (ABS(INTER_LOGIC.axisSpg_Vertical.velocity)) > (VERTICAL_SAFE_LIMIT*THRESHOLD) THEN
        VerticalOverride:= ((VERTICAL_SAFE_LIMIT*THRESHOLD)/(ABS(INTER_LOGIC.axisSpg_Vertical.velocity)))*NON_LINEAR_FUDGE_FACTOR;
        bTest := TRUE;
    ELSE
        VerticalOverride:= 1;//No vertical limiting required
        bTest := FALSE;
	END_IF
    
    IF (ABS(INTER_LOGIC.axisSpg_Horizontal.velocity)) > (HORIZONTAL_SAFE_LIMIT*THRESHOLD) THEN
        HorizontalOverride:= ((HORIZONTAL_SAFE_LIMIT*THRESHOLD)/(ABS(INTER_LOGIC.axisSpg_Horizontal.velocity)))*NON_LINEAR_FUDGE_FACTOR;
    ELSE
        HorizontalOverride:= 1;//No vertical limiting required
	END_IF
    
    IF (ABS(INTER_LOGIC.axisSpg_Rot.velocity)) > (ROTATION_SAFE_LIMIT*THRESHOLD) THEN
        RotationOverride:= (ROTATION_SAFE_LIMIT*THRESHOLD)/(ABS(INTER_LOGIC.axisSpg_Rot.velocity)); //*LOCALMODE_SPEED_OVERRIDE was removed from all of these for similar reasons, it should already be applied
    ELSE
        RotationOverride:= 1;//No vertical limiting required
	END_IF       
    
    SPEED_OVERRIDE_MODIFIER:= MIN(VerticalOverride, HorizontalOverride, RotationOverride);  //Take the worst case scenario
    
    FOR i:=1 TO INTER_LOGIC.ARRAYSIZE_ALLVIRTUALS DO
        astAxes[INTER_LOGIC.aVirtualAxisDefaults[i].axisID].stConfig.fOverride := LOCALMODE_SPEED_OVERRIDE * SPEED_OVERRIDE_MODIFIER;
        GVL_INTER.SPEED_LIMITING:= TRUE;
	END_FOR
END_IF

IF SPEED_OVERRIDE_MODIFIER < 1 THEN
    GVL_INTER.SPEED_LIMITING:= TRUE;
ELSE
    GVL_INTER.SPEED_LIMITING:= FALSE;
END_IF

END_PROGRAM

// ---- POUs/Application_Specific/Axes/Slit_North.TcPOU
PROGRAM Slit_North
VAR
//Outputs: Power for Limit switches, Home Sensors, etc.
    //bPowerSwitchesAxis1 AT %Q*: BOOL:= TRUE;

//Hardware interlocks
    //bInterlockFwdOK AT %I*: BOOL;
END_VAR

//Initial parameters of an Axis
IF _TaskInfo[fbGetCurTaskIndex.index].FirstCycle THEN
    //Initial default values:
    GVL.astAxes[AXIS_SLIT_NORTH].stConfig.eHomeSeq := E_HomingRoutines.eHomeToLimit_Fwd;
    GVL.astAxes[AXIS_SLIT_NORTH].stConfig.fHomePosition := 70.0;
    GVL.astAxes[AXIS_SLIT_NORTH].stConfig.fHomeFinishDistance := -5.0;
    GVL.astAxes[AXIS_SLIT_NORTH].stConfig.eRestorePosition := E_RestorePosition.eRestoreWithoutHome;
END_IF

//Define ACTIONS() or write exclusive code for an specific axis.
(*Eg. Stop when temperature reaches certain values, reduce speed if  a signal is activated, etc.
Eg. GVL.astAxes[x].stControl.bInterlockFwd := NOT bInterlockFwdOK;*)
astAxes[AXIS_SLIT_NORTH].stControl.bEnable:=TRUE;

END_PROGRAM

// ---- POUs/Application_Specific/Axes/Slit_South.TcPOU
PROGRAM Slit_South
VAR
//Outputs: Power for Limit switches, Home Sensors, etc.
    //bPowerSwitchesAxis1 AT %Q*: BOOL:= TRUE;

//Hardware interlocks
    //bInterlockFwdOK AT %I*: BOOL;
END_VAR

//Initial parameters of an Axis
IF _TaskInfo[fbGetCurTaskIndex.index].FirstCycle THEN
    //Initial default values:
    GVL.astAxes[AXIS_SLIT_SOUTH].stConfig.eHomeSeq := E_HomingRoutines.eHomeToLimit_Fwd;
    GVL.astAxes[AXIS_SLIT_SOUTH].stConfig.fHomePosition := 70.0;
    GVL.astAxes[AXIS_SLIT_SOUTH].stConfig.fHomeFinishDistance := -5.0;
    GVL.astAxes[AXIS_SLIT_SOUTH].stConfig.eRestorePosition := E_RestorePosition.eRestoreWithoutHome;
END_IF

//Define ACTIONS() or write exclusive code for an specific axis.
(*Eg. Stop when temperature reaches certain values, reduce speed if  a signal is activated, etc.
Eg. GVL.astAxes[x].stControl.bInterlockFwd := NOT bInterlockFwdOK;*)
astAxes[AXIS_SLIT_SOUTH].stControl.bEnable:=TRUE;

END_PROGRAM

// ---- POUs/Application_Specific/Axes/Slit_East.TcPOU
PROGRAM Slit_East
VAR
//Outputs: Power for Limit switches, Home Sensors, etc.
    //bPowerSwitchesAxis1 AT %Q*: BOOL:= TRUE;

//Hardware interlocks
    //bInterlockFwdOK AT %I*: BOOL;
END_VAR

//Initial parameters of an Axis
IF _TaskInfo[fbGetCurTaskIndex.index].FirstCycle THEN
    //Initial default values:
    GVL.astAxes[AXIS_SLIT_EAST].stConfig.eHomeSeq := E_HomingRoutines.eHomeToLimit_Fwd;
    GVL.astAxes[AXIS_SLIT_EAST].stConfig.fHomePosition := 70.0;
    GVL.astAxes[AXIS_SLIT_EAST].stConfig.fHomeFinishDistance := -5.0;
    GVL.astAxes[AXIS_SLIT_EAST].stConfig.eRestorePosition := E_RestorePosition.eRestoreWithoutHome;
END_IF

//Define ACTIONS() or write exclusive code for an specific axis.
(*Eg. Stop when temperature reaches certain values, reduce speed if  a signal is activated, etc.
Eg. GVL.astAxes[x].stControl.bInterlockFwd := NOT bInterlockFwdOK;*)
astAxes[AXIS_SLIT_EAST].stControl.bEnable:=TRUE;

END_PROGRAM

// ---- POUs/Application_Specific/Axes/Slit_West.TcPOU
PROGRAM Slit_West
VAR
//Outputs: Power for Limit switches, Home Sensors, etc.
    //bPowerSwitchesAxis1 AT %Q*: BOOL:= TRUE;

//Hardware interlocks
    //bInterlockFwdOK AT %I*: BOOL;
END_VAR

//Initial parameters of an Axis
IF _TaskInfo[fbGetCurTaskIndex.index].FirstCycle THEN
    //Initial default values:
    GVL.astAxes[AXIS_SLIT_WEST].stConfig.eHomeSeq := E_HomingRoutines.eHomeToLimit_Fwd;
    GVL.astAxes[AXIS_SLIT_WEST].stConfig.fHomePosition := 70.0;
    GVL.astAxes[AXIS_SLIT_WEST].stConfig.fHomeFinishDistance := -5.0;
    GVL.astAxes[AXIS_SLIT_WEST].stConfig.eRestorePosition := E_RestorePosition.eRestoreWithoutHome;
END_IF

//Define ACTIONS() or write exclusive code for an specific axis.
(*Eg. Stop when temperature reaches certain values, reduce speed if  a signal is activated, etc.
Eg. GVL.astAxes[x].stControl.bInterlockFwd := NOT bInterlockFwdOK;*)
astAxes[AXIS_SLIT_WEST].stControl.bEnable:=TRUE;

END_PROGRAM

// ---- POUs/Application_Specific/Applications/Slit_3.TcPOU
PROGRAM Slit_3
VAR
    NorthSouthPowerOutput AT %Q* : BOOL:= TRUE;
    EastWestPowerOutput AT %Q* : BOOL:= TRUE;
END_VAR

END_PROGRAM

// ---- POUs/Application_Specific/Applications/Inclinometer.TcPOU
PROGRAM Inclinometer
VAR
    INC_VAL AT%I* : UINT;
    INC_VAL_LINEAR_SCALED : LREAL;
    MEASURED_UPPER_LIMIT : LREAL := 32767;
    MEASURED_LOWER_LIMIT : LREAL := 0;
    DESIRED_UPPER_LIMIT_LINEAR : LREAL := 1;
    DESIRED_LOWER_LIMIT_LINEAR : LREAL := -1;
    DESIRED_UPPER_LIMIT_SF : LREAL := 20;
    DESIRED_LOWER_LIMIT_SF : LREAL := 4;
    INC_VAL_SF_SCALED : LREAL;
    INC_VAL_DATASHEET_SCALED : LREAL;
    SCALE_FACTOR_DS : LREAL := 458.39;
 
END_VAR

INC_VAL_LINEAR_SCALED := DESIRED_LOWER_LIMIT_LINEAR + (DESIRED_UPPER_LIMIT_LINEAR - DESIRED_LOWER_LIMIT_LINEAR)*((UINT_TO_LREAL(INC_VAL) - MEASURED_LOWER_LIMIT)/(MEASURED_UPPER_LIMIT - MEASURED_LOWER_LIMIT));
 
INC_VAL_SF_SCALED := DESIRED_LOWER_LIMIT_SF + (DESIRED_UPPER_LIMIT_SF - DESIRED_LOWER_LIMIT_SF)*((UINT_TO_LREAL(INC_VAL) - MEASURED_LOWER_LIMIT)/(MEASURED_UPPER_LIMIT - MEASURED_LOWER_LIMIT));
INC_VAL_DATASHEET_SCALED := RAD_TO_DEG(ASIN((INC_VAL_SF_SCALED-12)/SCALE_FACTOR_DS));
GVL_INTER.INCLINOMETER_ANGLE:= INC_VAL_LINEAR_SCALED;

END_PROGRAM

// ---- POUs/Application_Specific/Applications/SBT_CODE_notused.TcPOU
PROGRAM SBT_CODE_notused
VAR
	iStep: INT;
	bTriggerBrakeTest: BOOL;
	bError: BOOL;
	bBusy : BOOL;
	bErrorCode: STRING;
	fbBrakeControl : FB_CoEAX8000BrakeControl;
	Axis1 : AXIS_REF;
	Timer : TON;
	ErrorAck: BOOL;
	fbReset : MC_Reset; (*Unsure if this is correct FB but I think it is*)
	ChA_StartBrakeTest: BOOL;
	bOutputStageSafetyState: BYTE; (*Input*)
	MCPower : MC_Power;
	fbAX8000BrakeTest : FB_CoEAX8000BrakeTest;
	ChA_TestSucceeded: BOOL;
	ChA_BrakeTestPassed: BOOL;
    
    
END_VAR

Axis1.ReadStatus();
CASE iStep OF
	
	0:	(*TriggerBrakeTest*)		
			IF bTriggerBrakeTest THEN
				bTriggerBrakeTest := FALSE;
				iStep := 10;
				bError := FALSE;
				bErrorCode := '';
				ChA_StartBrakeTest := TRUE;
			END_IF
			
			
	10:	(*CloseBrake*)
		fbBrakeControl(		(*FB_CoEAX8000BrakeControl*)
			Axis := Axis1,
			Execute := TRUE,
			Mode := E_AX8000BrakeMode.eAX8000BrakeMode_Lock );

		IF NOT fbBrakeControl.Busy AND NOT fbBrakeControl.Error THEN
			fbBrakeControl(Axis:= Axis1, Execute := FALSE, Mode := E_AX8000BrakeMode.eAX8000BrakeMode_Lock);
		ELSIF NOT fbBrakeControl.Busy AND fbBrakeControl.Error THEN
			fbBrakeControl(Axis:= Axis1, Execute := FALSE, Mode := E_AX8000BrakeMode.eAX8000BrakeMode_Lock);
			bBusy := FALSE;
			bError := TRUE;
			bErrorCode := 'CloseBrakeFailed';
			iStep := 0;
		END_IF
		
		
	20: (*Time which is required in order to close the brake*)
		Timer(IN := TRUE, PT := T#100MS, Q => , ET=> );
			
		IF Timer.Q THEN
			Timer(IN := FALSE);
			iStep := 30;
		END_IF
	
		
	30: (*Send reset to E-Stop FB inside safety project --> final STO release*)
		ErrorAck := TRUE;
		Timer(IN := TRUE, PT := T#500MS);
		
		IF Timer.Q THEN
			ErrorAck := FALSE;
			Timer(IN := FALSE);
			iStep := 40;
		END_IF
	
		
	40: (*Send reset --> in case NC or drive has an error*)
		IF Axis1.Status.Error THEN
			fbReset(
				Axis:= Axis1,
				Execute := TRUE);
		ELSE
			iStep := 50;
		END_IF
		
		IF fbReset.Done THEN
			fbReset(Axis:= Axis1, Execute := FALSE);
			iStep := 50;
		ELSIF NOT fbReset.Busy AND fbReset.Error THEN
			fbReset(Axis:= Axis1, Execute := FALSE);
			bError := TRUE;
			bErrorCode := 'NC-AxisResetFailed';
			ChA_StartBrakeTest := FALSE;
			iStep := 999;
		END_IF
	
		
	50: (*Check if outputstage is blocked via STO*)
		IF bOutputStageSafetyState.0 THEN
			iStep := 60;
			Timer(IN := FALSE);
		ELSE
			iStep := 30;
		END_IF
		
		
	60: (*Enable Motor*)
		MCPower(
			Axis := Axis1,
			Enable := TRUE,
			Enable_Positive := TRUE,
			Enable_Negative := TRUE,
			Override := 100);
			
		IF MCPower.Status THEN
			iStep := 70;
		ELSIF McPower.Error THEN
			iStep := 999;
			bError := TRUE;
			bErrorCode := 'EnableAxisFailed';
			ChA_StartBrakeTest := FALSE;
		END_IF
		
		
		
	70: (*FB_CoEAX8000BrakeTest*)
		fbAX8000BrakeTest(
			Axis := Axis1,
			Execute := TRUE,
			Succeeded := ChA_TestSucceeded,
			Torque := 0.5,
			VelocityLimit := 100,
			Timeout := T#10S,
			Busy => ,
			Error => ,
			ErrorID => );
			
		IF NOT fbAX8000BrakeTest.Busy AND NOT fbAX8000BrakeTest.Error THEN			
			fbAX8000BrakeTest(Axis := Axis1 , Execute := FALSE);
			iStep := 80;
		ELSIF NOT fbAX8000BrakeTest.Busy AND fbAX8000BrakeTest.Error THEN
			fbAX8000BrakeTest(Axis := Axis1 , Execute := FALSE);
			bError := TRUE;
			bErrorCode := 'FB_BrakeTestSendError';
			iStep := 80;
		END_IF
		
		
	80: (*Switch off ChA_StartBrakeTest*)
		Timer(IN := TRUE, PT := T#1S);
		
		IF ChA_BrakeTestPassed THEN
			ChA_StartBrakeTest := FALSE;
			Timer(IN := FALSE);
			iStep := 90;
		END_IF
		
		IF Timer.Q THEN
			Timer(IN := FALSE);
			ChA_StartBrakeTest := FALSE;
			iStep := 90;
		END_IF
		
		
	90: (*Switch Brake to automatic*)
		fbBrakeControl(
			Axis := Axis1,
			Execute := TRUE,
			Mode := E_AX8000BrakeMode.eAX8000BrakeMode_Automatic);
			
		IF NOT fbBrakeControl.Busy AND NOT fbBrakeControl.Error THEN
			fbBrakeControl(Axis := Axis1, Execute := FALSE, Mode := E_AX8000BrakeMode.eAX8000BrakeMode_Lock);
			iStep := 100;
		ELSIF NOT fbBrakeControl.Busy AND fbBrakeControl.Error THEN
			fbBrakeControl(Axis := Axis1, Execute := FALSE, Mode := E_AX8000BrakeMode.eAX8000BrakeMode_Lock);
			bBusy := FALSE;
			bError := TRUE;
			bErrorCode := 'SwitchBrakeToAutomaticFailed';
			iStep := 0;
		END_IF
	
	
	100: (*Disable Motor*)
		MCPower(
			Axis := Axis1,
			Enable := FALSE,
			Enable_Positive := FALSE,
			Enable_Negative := FALSE,
			Override := 0);	

		IF NOT MCPower.Status THEN
			iStep := 0;
		END_IF
		
		
	999:
		MCPower(
			Axis := Axis1,
			Enable := FALSE,
			Enable_Positive := FALSE,
			Enable_Negative := FALSE,
			Override := 0);	
		
		fbReset(
			Axis:= Axis1,
			Execute := TRUE,
			Done => ,
			Busy => ,
			Error => ,
			ErrorID => );
		
		IF fbReset.Done THEN
			iStep := 0;
			fbReset(Axis:= Axis1, Execute := FALSE);
			ChA_StartBrakeTest := FALSE;
		ELSIF NOT fbReset.Busy AND fbReset.Error THEN
			fbReset(Axis:= Axis1, Execute := FALSE);
			bError := TRUE;
			bErrorCode := 'NC-Axis reset failed';
			ChA_StartBrakeTest := FALSE;
			iStep := 0;
		END_IF
END_CASE

END_PROGRAM

// ---- tc_mca_std_lib/POUs/FB_ESSMonitoring.TcPOU

FUNCTION_BLOCK FB_ESSMonitoring
VAR_INPUT
    nEcMasterNetId: T_AmsNetId;
END_VAR
VAR_OUTPUT
    aErrorID: ARRAY [1..nMaxAlarms] OF INT;
    aErrorMsg: ARRAY [1..nMaxAlarms] OF STRING;
    nEcMasterFramesLost: UDINT;
    nCPULoad: UDINT;
    fCycleExecTime_ms: REAL;
    nAlarmGrpBitNumber: UDINT;
END_VAR
VAR
    //Outputs
    bFan1 AT %Q*: BOOL := TRUE;
    bFan2 AT %Q*: BOOL := TRUE;
    bDCSupplyLED AT %Q*: BOOL;
    bAcknowledgeLED AT %Q*: BOOL;
    bStatusLED AT %Q*: BOOL;
    bWarningLED AT %Q*: BOOL;
    bEmergencyLED AT %Q*: BOOL;
    //Inputs
    b24VDC1_OK AT %I*: BOOL;
    b24VDC2_OK AT %I*: BOOL;
    b48VDC1_OK AT %I*: BOOL;
    bFuse1_OK AT %I*: BOOL;
    bFuse2_OK AT %I*: BOOL;
    bFuse3_OK AT %I*: BOOL;
    bFuse4_OK AT %I*: BOOL;
    bFuse5_OK AT %I*: BOOL;
    bFuse6_OK AT %I*: BOOL;
    bFuse7_OK AT %I*: BOOL;
    bFuse8_OK AT %I*: BOOL;
    bSafety_OK AT %I*: BOOL;
    bFan1_OK AT %I*: BOOL;
    bFan2_OK AT %I*: BOOL;
    nTemp1 AT %I*: INT;
    nTemp2 AT %I*: INT;
    nEcMasterDevState AT %I*: UINT;
    aAlarmList: ARRAY [1..nMaxAlarms] OF ST_MonitoringAlarm := [
                    (*[1]*)(nStatusLED:=E_MonitoringLedFunction.eFast, nWarningLED:=E_MonitoringLedFunction.eUndefined, nEmergencyLED:=E_MonitoringLedFunction.eSteady, nAcknowledgeLED:=E_MonitoringLedFunction.eUndefined, nErrorID:=1 ,sErrorMsg:='The DC OK Status from PS or DC-DC converter 24V-1 is OFF.'),
                    (*[2]*)(nStatusLED:=E_MonitoringLedFunction.eUndefined, nWarningLED:=E_MonitoringLedFunction.eUndefined, nEmergencyLED:=E_MonitoringLedFunction.eUndefined, nAcknowledgeLED:=E_MonitoringLedFunction.eUndefined, nErrorID:=2 ,sErrorMsg:='The DC OK Status from PS 24V-2 is OFF.'),
                    (*[3]*)(nStatusLED:=E_MonitoringLedFunction.eFast, nWarningLED:=E_MonitoringLedFunction.eUndefined, nEmergencyLED:=E_MonitoringLedFunction.eSteady, nAcknowledgeLED:=E_MonitoringLedFunction.eUndefined, nErrorID:=4 ,sErrorMsg:='The DC OK Status from PS 48V-1 is OFF.'),
                    (*[4]*)(nStatusLED:=E_MonitoringLedFunction.eUndefined, nWarningLED:=E_MonitoringLedFunction.eUndefined, nEmergencyLED:=E_MonitoringLedFunction.eUndefined, nAcknowledgeLED:=E_MonitoringLedFunction.eUndefined, nErrorID:=8 ,sErrorMsg:='Output 1 on LOCC box 1 tripped'),
                    (*[5]*)(nStatusLED:=E_MonitoringLedFunction.eSlow, nWarningLED:=E_MonitoringLedFunction.eUndefined, nEmergencyLED:=E_MonitoringLedFunction.eSteady, nAcknowledgeLED:=E_MonitoringLedFunction.eUndefined, nErrorID:=9 ,sErrorMsg:='Output 2 on LOCC box 1 tripped'),
                    (*[6]*)(nStatusLED:=E_MonitoringLedFunction.eUndefined, nWarningLED:=E_MonitoringLedFunction.eUndefined, nEmergencyLED:=E_MonitoringLedFunction.eUndefined, nAcknowledgeLED:=E_MonitoringLedFunction.eUndefined, nErrorID:=10 ,sErrorMsg:='Output 1 on LOCC box 2 tripped'),
                    (*[7]*)(nStatusLED:=E_MonitoringLedFunction.eSlow, nWarningLED:=E_MonitoringLedFunction.eUndefined, nEmergencyLED:=E_MonitoringLedFunction.eSteady, nAcknowledgeLED:=E_MonitoringLedFunction.eUndefined, nErrorID:=11 ,sErrorMsg:='Output 2 on LOCC box 2 tripped'),
                    (*[8]*)(nStatusLED:=E_MonitoringLedFunction.eSteady, nWarningLED:=E_MonitoringLedFunction.eSteady, nEmergencyLED:=E_MonitoringLedFunction.eUndefined, nAcknowledgeLED:=E_MonitoringLedFunction.eUndefined, nErrorID:=12 ,sErrorMsg:='Output 1 on LOCC box 3 tripped'),
                    (*[9]*)(nStatusLED:=E_MonitoringLedFunction.eSteady, nWarningLED:=E_MonitoringLedFunction.eSteady, nEmergencyLED:=E_MonitoringLedFunction.eUndefined, nAcknowledgeLED:=E_MonitoringLedFunction.eUndefined, nErrorID:=13 ,sErrorMsg:='Output 2 on LOCC box 3 tripped'),
                    (*[10]*)(nStatusLED:=E_MonitoringLedFunction.eSlow, nWarningLED:=E_MonitoringLedFunction.eSteady, nEmergencyLED:=E_MonitoringLedFunction.eUndefined, nAcknowledgeLED:=E_MonitoringLedFunction.eUndefined, nErrorID:=14 ,sErrorMsg:='LOCC box 4 or single DC breaker 1 tripped'),
                    (*[11]*)(nStatusLED:=E_MonitoringLedFunction.eSlow, nWarningLED:=E_MonitoringLedFunction.eSteady, nEmergencyLED:=E_MonitoringLedFunction.eUndefined, nAcknowledgeLED:=E_MonitoringLedFunction.eUndefined, nErrorID:=15 ,sErrorMsg:='LOCC box 5 or single DC breaker 2 tripped'),
                    (*[12]*)(nStatusLED:=E_MonitoringLedFunction.eUndefined, nWarningLED:=E_MonitoringLedFunction.eSteady, nEmergencyLED:=E_MonitoringLedFunction.eUndefined, nAcknowledgeLED:=E_MonitoringLedFunction.eUndefined, nErrorID:=21 ,sErrorMsg:='Speed of Fan 1 below a critical limit'),
                    (*[13]*)(nStatusLED:=E_MonitoringLedFunction.eUndefined, nWarningLED:=E_MonitoringLedFunction.eSteady, nEmergencyLED:=E_MonitoringLedFunction.eUndefined, nAcknowledgeLED:=E_MonitoringLedFunction.eUndefined, nErrorID:=22 ,sErrorMsg:='Speed of Fan 2 below a critical limit'),
                    (*[14]*)(nStatusLED:=E_MonitoringLedFunction.eUndefined, nWarningLED:=E_MonitoringLedFunction.eSteady, nEmergencyLED:=E_MonitoringLedFunction.eSteady, nAcknowledgeLED:=E_MonitoringLedFunction.eUndefined, nErrorID:=23 ,sErrorMsg:='Temperature 1 too high' ),
                    (*[15]*)(nStatusLED:=E_MonitoringLedFunction.eUndefined, nWarningLED:=E_MonitoringLedFunction.eSteady, nEmergencyLED:=E_MonitoringLedFunction.eSteady, nAcknowledgeLED:=E_MonitoringLedFunction.eUndefined, nErrorID:=24 ,sErrorMsg:='Temperature 2 too high'),
                    (*[16]*)(nStatusLED:=E_MonitoringLedFunction.eSteady, nWarningLED:=E_MonitoringLedFunction.eSteady, nEmergencyLED:=E_MonitoringLedFunction.eUndefined, nAcknowledgeLED:=E_MonitoringLedFunction.eUndefined, nErrorID:=30 ,sErrorMsg:='Safety relay 1 triggered'),
                    (*[17]*)(nStatusLED:=E_MonitoringLedFunction.eSteady, nWarningLED:=E_MonitoringLedFunction.eSlow, nEmergencyLED:=E_MonitoringLedFunction.eUndefined, nAcknowledgeLED:=E_MonitoringLedFunction.eUndefined, nErrorID:=101 ,sErrorMsg:='EtherCAT Master is not ok'),
                    (*[18]*)(nStatusLED:=E_MonitoringLedFunction.eSteady, nWarningLED:=E_MonitoringLedFunction.eSlow, nEmergencyLED:=E_MonitoringLedFunction.eSteady, nAcknowledgeLED:=E_MonitoringLedFunction.eUndefined, nErrorID:=102 ,sErrorMsg:='At least one EtherCAT slave is not in OP state'),
                    (*[19]*)(nStatusLED:=E_MonitoringLedFunction.eSteady, nWarningLED:=E_MonitoringLedFunction.eSlow, nEmergencyLED:=E_MonitoringLedFunction.eSteady, nAcknowledgeLED:=E_MonitoringLedFunction.eUndefined, nErrorID:=103 ,sErrorMsg:='At least one EtherCAT slave link is faulted'),
                    (*[20]*)(nStatusLED:=E_MonitoringLedFunction.eSteady, nWarningLED:=E_MonitoringLedFunction.eSlow, nEmergencyLED:=E_MonitoringLedFunction.eUndefined, nAcknowledgeLED:=E_MonitoringLedFunction.eUndefined, nErrorID:=104 ,sErrorMsg:='Overflow in PLC cycle time'),
                    (*[21]*)(nStatusLED:=E_MonitoringLedFunction.eSteady, nWarningLED:=E_MonitoringLedFunction.eSlow, nEmergencyLED:=E_MonitoringLedFunction.eUndefined, nAcknowledgeLED:=E_MonitoringLedFunction.eUndefined, nErrorID:=105 ,sErrorMsg:='CPU Load High')];

    aTempErrorID: ARRAY [1..nMaxAlarms] OF INT;
    aTempErrorMsg: ARRAY [1..nMaxAlarms] OF STRING;
    nLEDAlarmID: INT;
    sLEDAlarmMsg: STRING;
    nAlarmCnt: INT;
    nAlarmBitNumber: UDINT;

    bCPUOverloaded: BOOL;
    bEcMasterNotOK: BOOL;
    bSlaveStateNotOP: BOOL;
    bSlaveLinkNotOK: BOOL;
    bCycleTimeExceeded: BOOL;
    //Cpu Monitor
    fbMonitorCPU: TC_CpuUsage;
    fbUpdateCPULoadTON: TON;
    fMaxCPULoad: USINT := 85;
    //Ehtercat master device state
    bEcLinkError: BOOL;
    bEcIOlocked: BOOL;
    bEcLinkErrorRedundancyAdapter: BOOL;
    bEcMissingFrame: BOOL;
    bEcOutofSendResources: BOOL;
    bEcWatchdogTriggered: BOOL;
    bEcEthernetDriverNotFound: BOOL;
    bEcIOresetActive: BOOL;
    bEcSlaveINIT: BOOL;
    bEcSlavePreOP: BOOL;
    bEcSlaveSafeOP: BOOL;
    bEcSlaveError: BOOL;
    bEcDCnotInSync: BOOL;
    //Ehtercat slave device state
    fbUpdateEcSlaveStateTON: TON;
    fbGetEcSlaveStates: FB_EcGetAllSlaveStates;
    stSlaveState: ARRAY[0..nMaxECSlaves] OF ST_EcSlaveState;
    nActualEcSlaves: INT := 0;
    i: INT;
    //Frame statistics
    fbUpdateEcMasterFrame: TON;
    fbGetEcMasterFrames: FB_EcMasterFrameStatistic;

    nAcknowledgeLED: E_MonitoringLedFunction;
    nStatusLED: E_MonitoringLedFunction;
    nWarningLED: E_MonitoringLedFunction;
    nEmergencyLED: E_MonitoringLedFunction;
    fbFastBlinkOn: TON;
    fbFastBlinkOff: TON;
    bFastBlink: BOOL;
    fbSlowBlinkOn: TON;
    fbSlowBlinkOff: TON;
    bSlowBlink: BOOL;
END_VAR
VAR CONSTANT
    nMaxAlarms: INT := 50;
    nMaxECSlaves: INT := 255;
    nMaxTemp: INT := 10000;
END_VAR


actMonitorAlarms();
actMonitorCPU();
actMonitorEtherCAT();

ACTION actMonitorAlarms:

aAlarmList[1].bAlarmSet := NOT b24VDC1_OK;
aAlarmList[1].bAlarmReset:= TRUE;
aAlarmList[2].bAlarmSet := b24VDC2_OK;
aAlarmList[2].bAlarmReset:= TRUE;
aAlarmList[3].bAlarmSet := NOT b48VDC1_OK;
aAlarmList[3].bAlarmReset:= TRUE;
aAlarmList[4].bAlarmSet := bFuse1_OK;
aAlarmList[4].bAlarmReset:= TRUE;
aAlarmList[5].bAlarmSet :=  bFuse2_OK;
aAlarmList[5].bAlarmReset:= TRUE;
aAlarmList[6].bAlarmSet := bFuse3_OK;
aAlarmList[6].bAlarmReset:= TRUE;
aAlarmList[7].bAlarmSet := bFuse4_OK;
aAlarmList[7].bAlarmReset:= TRUE;
aAlarmList[8].bAlarmSet := bFuse5_OK;
aAlarmList[8].bAlarmReset:= TRUE;
aAlarmList[9].bAlarmSet := bFuse6_OK;
aAlarmList[9].bAlarmReset:= TRUE;
aAlarmList[10].bAlarmSet := bFuse7_OK;
aAlarmList[10].bAlarmReset:= TRUE;
aAlarmList[11].bAlarmSet := bFuse8_OK;
aAlarmList[11].bAlarmReset:= TRUE;
aAlarmList[12].bAlarmSet := NOT bFan1_OK;
aAlarmList[12].bAlarmReset:= TRUE;
aAlarmList[13].bAlarmSet := NOT bFan2_OK;
aAlarmList[13].bAlarmReset:= TRUE;
aAlarmList[14].bAlarmSet := nTemp1 > nMaxTemp;
aAlarmList[14].bAlarmReset:= TRUE;
aAlarmList[15].bAlarmSet := nTemp2 > nMaxTemp;
aAlarmList[15].bAlarmReset:= TRUE;
aAlarmList[16].bAlarmSet := NOT bSafety_OK;
aAlarmList[16].bAlarmReset:= TRUE;
aAlarmList[17].bAlarmSet := bEcMasterNotOK;
aAlarmList[17].bAlarmReset:= TRUE;
aAlarmList[18].bAlarmSet := bSlaveStateNotOP;
aAlarmList[18].bAlarmReset:= TRUE;
aAlarmList[19].bAlarmSet := bSlaveLinkNotOK;
aAlarmList[19].bAlarmReset:= TRUE;
aAlarmList[20].bAlarmSet := bCycleTimeExceeded;
aAlarmList[20].bAlarmReset:= TRUE;
aAlarmList[21].bAlarmSet := bCPUOverloaded;
aAlarmList[21].bAlarmReset:= TRUE;

FOR i:=1 TO nMaxAlarms DO
    mAlarm(stAlarmData:= aAlarmList[i]);
    IF i = 1 THEN
        nAlarmCnt := 0;
        nAlarmBitNumber := 0;
        MEMSET(ADR(aTempErrorID), 0, SIZEOF(aTempErrorID));
        MEMSET(ADR(aTempErrorMsg), 0, SIZEOF(aTempErrorMsg));
    ELSIF i = nMaxAlarms THEN
        aErrorID := aTempErrorID;
        aErrorMsg := aTempErrorMsg;
        nAlarmGrpBitNumber := nAlarmBitNumber;
    END_IF

    IF aAlarmList[i].bAlarmActive THEN
        nAlarmCnt := nAlarmCnt + 1;
        aTempErrorID[nAlarmCnt] := aAlarmList[i].nErrorID;
        aTempErrorMsg[nAlarmCnt] := aAlarmList[i].sErrorMsg;
        IF nLEDAlarmID = 0 OR (nWarningLED = E_MonitoringLedFunction.eUndefined AND nEmergencyLED = E_MonitoringLedFunction.eUndefined AND aAlarmList[i].nWarningLED > E_MonitoringLedFunction.eUndefined) OR (nEmergencyLED = E_MonitoringLedFunction.eUndefined AND aAlarmList[i].nEmergencyLED > E_MonitoringLedFunction.eUndefined) THEN
            nLEDAlarmID := i;
            sLEDAlarmMsg := aAlarmList[i].sErrorMsg;
            nEmergencyLED := aAlarmList[i].nEmergencyLED;
            nWarningLED := aAlarmList[i].nWarningLED;
            nStatusLED := aAlarmList[i].nStatusLED;
            nAcknowledgeLED := aAlarmList[i].nAcknowledgeLED;
        END_IF
        CASE aAlarmList[i].nErrorID OF
            1,4:
            nAlarmBitNumber.0 := TRUE;
            9,12,13:
            nAlarmBitNumber.1 := TRUE;
            10,11:
            nAlarmBitNumber.2 := TRUE;
            14,15:
            nAlarmBitNumber.3 := TRUE;
            21,22:
            nAlarmBitNumber.4 := TRUE;
            23,24:
            nAlarmBitNumber.5 := TRUE;
            104,105:
            nAlarmBitNumber.6 := TRUE;
            103:
            nAlarmBitNumber.7 := TRUE;
            102:
            nAlarmBitNumber.8 := TRUE;
            30:
            nAlarmBitNumber.9 := TRUE;
        END_CASE
    ELSIF NOT aAlarmList[i].bAlarmActive THEN
        IF nLEDAlarmID = i THEN
            nLEDAlarmID := 0;
            sLEDAlarmMsg := '';
            nEmergencyLED := 0;
            nWarningLED := 0;
            nStatusLED := 0;
            nAcknowledgeLED := 0;
        END_IF
    END_IF
END_FOR

fbFastBlinkOn(IN:=NOT fbFastBlinkOff.q , PT:=T#250MS , Q=> , ET=> );
fbFastBlinkOff(IN:=fbFastBlinkOn.Q , PT:=T#250MS , Q=> , ET=> );
bFastBlink := fbFastBlinkOn.q;

fbSlowBlinkOn(IN:=NOT fbSlowBlinkOff.q , PT:=T#750MS , Q=> , ET=> );
fbSlowBlinkOff(IN:=fbSlowBlinkOn.Q , PT:=T#750MS , Q=> , ET=> );
bSlowBlink := fbSlowBlinkOn.q;

bEmergencyLED := (nEmergencyLED = E_MonitoringLedFunction.eSteady) OR (nEmergencyLED = E_MonitoringLedFunction.eFast AND bFastBlink) OR (nEmergencyLED = E_MonitoringLedFunction.eSlow AND bSlowBlink);
bWarningLED := (nWarningLED = E_MonitoringLedFunction.eSteady) OR (nWarningLED = E_MonitoringLedFunction.eFast AND bFastBlink) OR (nWarningLED = E_MonitoringLedFunction.eSlow AND bSlowBlink);
bStatusLED := (nStatusLED = E_MonitoringLedFunction.eSteady) OR (nStatusLED = E_MonitoringLedFunction.eFast AND bFastBlink) OR (nStatusLED = E_MonitoringLedFunction.eSlow AND bSlowBlink);
bAcknowledgeLED := (nAcknowledgeLED = E_MonitoringLedFunction.eSteady) OR (nAcknowledgeLED = E_MonitoringLedFunction.eFast AND bFastBlink) OR (nAcknowledgeLED = E_MonitoringLedFunction.eSlow AND bSlowBlink);
END_ACTION

ACTION actMonitorCPU:

//Cpu Monitor
fbUpdateCPULoadTON(IN:=NOT fbUpdateCPULoadTON.q , PT:=T#100MS , Q=> , ET=> );
fbMonitorCPU(START:=fbUpdateCPULoadTON.q, TMOUT:= T#5S);

bCPUOverloaded := fbMonitorCPU.USAGE > fMaxCPULoad;
nCPULoad := fbMonitorCPU.USAGE;

fCycleExecTime_ms := UDINT_TO_REAL(_TaskInfo[fbGetCurTaskIndex.index].LastExecTime) / 10000;
bCycleTimeExceeded := _TaskInfo[fbGetCurTaskIndex.index].CycleTimeExceeded;
END_ACTION

ACTION actMonitorEtherCAT:

//Read frames
fbUpdateEcMasterFrame(IN:=NOT fbUpdateEcMasterFrame.q , PT:=T#1000MS , Q=> , ET=> );
fbGetEcMasterFrames(sNetId:= nEcMasterNetId, bExecute:= fbUpdateEcMasterFrame.q);

nEcMasterFramesLost := fbGetEcMasterFrames.nLostFrames;


//Check ethercat slave device state
fbUpdateEcSlaveStateTON(IN:=NOT fbUpdateEcSlaveStateTON.q , PT:=T#100MS , Q=> , ET=> );
fbGetEcSlaveStates(sNetId:= nEcMasterNetId, pStateBuf := ADR(stSlaveState), cbBufLen:=SIZEOF(stSlaveState), bExecute:=fbUpdateEcSlaveStateTON.q);
nActualEcSlaves:=UINT_TO_INT(fbGetEcSlaveStates.nSlaves);

FOR i:=0 TO nActualEcSlaves-1 DO
    IF i = 0 THEN
        bSlaveStateNotOP := FALSE;
        bSlaveLinkNotOK := FALSE;
    END_IF
    IF stSlaveState[i].deviceState <> EC_DEVICE_STATE_OP THEN
        bSlaveStateNotOP := TRUE;
    END_IF
    IF stSlaveState[i].linkState <> EC_LINK_STATE_OK THEN
        bSlaveLinkNotOK := TRUE;
    END_IF
END_FOR

//Check ethercat master device state
bEcLinkError := nEcMasterDevState.0;
bEcIOlocked := nEcMasterDevState.1;
bEcLinkErrorRedundancyAdapter := nEcMasterDevState.2;
bEcMissingFrame := nEcMasterDevState.3;
bEcOutofSendResources := nEcMasterDevState.4;
bEcWatchdogTriggered := nEcMasterDevState.5;
bEcEthernetDriverNotFound := nEcMasterDevState.6;
bEcIOresetActive := nEcMasterDevState.7;
bEcSlaveINIT := nEcMasterDevState.8;
bEcSlavePreOP := nEcMasterDevState.9;
bEcSlaveSafeOP := nEcMasterDevState.10;
bEcSlaveError := nEcMasterDevState.11;
bEcDCnotInSync := nEcMasterDevState.12;

bEcMasterNotOK := nEcMasterDevState > 0;
END_ACTION


METHOD mAlarm : BOOL
VAR_IN_OUT
    stAlarmData: ST_MonitoringAlarm;
END_VAR

IF stAlarmData.bAlarmSet THEN
    stAlarmData.bAlarmActive := TRUE;
ELSIF stAlarmData.bAlarmReset THEN
    stAlarmData.bAlarmActive := FALSE;
END_IF
END_METHOD

END_FUNCTION_BLOCK

// ---- tc_mca_std_lib/VISUs/MainVisu.TcVIS
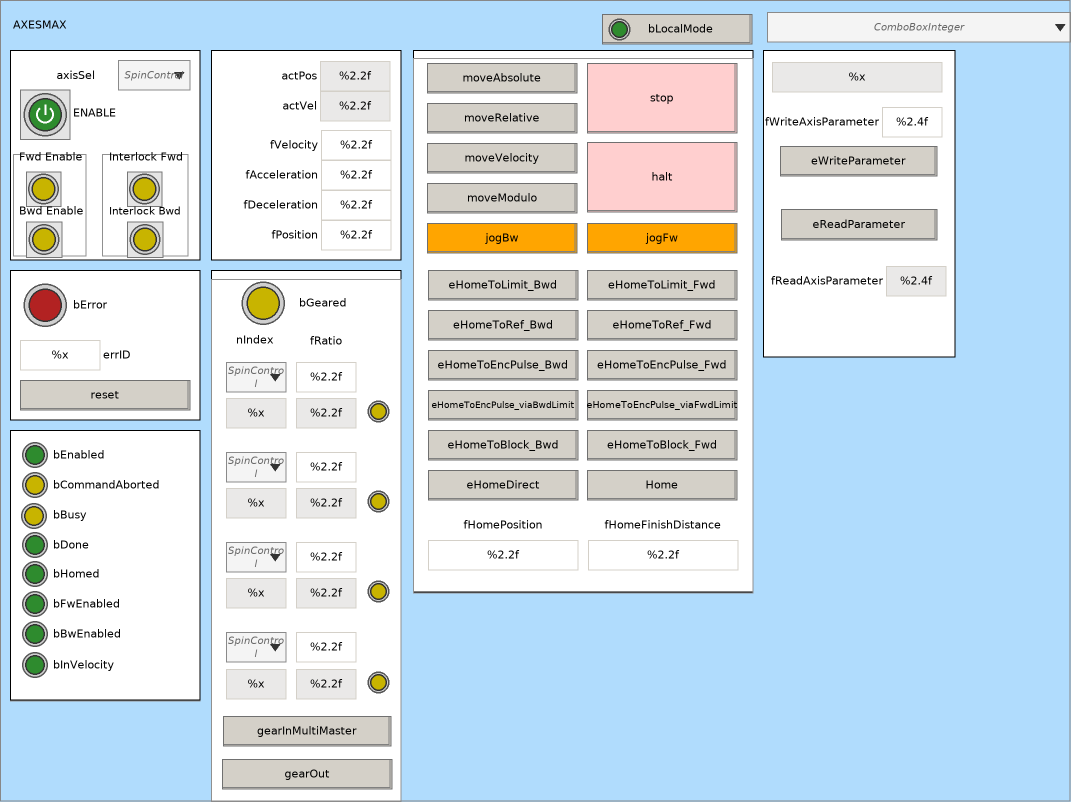
VISUALIZATION MainVisu  // 1071x802
    Rectangle (413,50 340x542)
    GroupBox (413,50 340x543)
        Button (174,92 150x70), "halt", pressed state: GVL.astAxes[Main.hmiAxisSelection].stControl.bHalt, input disabled if: GVL.astAxes[MAIN.hmiAxisSelection].stStatus.bGeared, text list: "languageSupport", text index: "halt"
            toggle GVL.astAxes[Main.hmiAxisSelection].stControl.bHalt
        Button (174,420 150x30), "Home", input disabled if: GVL.astAxes[MAIN.hmiAxisSelection].stStatus.bGeared, text list: 'languageSupport', text index: "Home"
            OnMouseClick: execute { GVL.astAxes[Main.hmiAxisSelection].stControl.eCommand:=E_MotionFunctions.eHome; GVL.astAxes[Main.hmiAxisSelection].stControl.bExecute:=TRUE; }
        Button (15,380 150x30), "eHomeToBlock_Bwd", input disabled if: GVL.astAxes[MAIN.hmiAxisSelection].stStatus.bGeared, text list: 'languageSupport', text index: "eHomeToBlock_Bwd"
            OnMouseClick: execute {
                GVL.astAxes[Main.hmiAxisSelection].stControl.eCommand:=E_MotionFunctions.eHome;
                GVL.astAxes[Main.hmiAxisSelection].stConfig.eHomeSeq:=E_HomingRoutines.eHomeToBlock_Bwd;
                GVL.astAxes[Main.hmiAxisSelection].stControl.bExecute:=TRUE;
            }
    Rectangle (211,270 190x531)
    GroupBox (211,271 190x531)
        SpinControl (15,91 60x30), variable: GVL.astAxes[MAIN.hmiAxisSelection].stConfig.astMultiMasterAxis[1].nIndex
            p651134158: GVL_APP.nAXIS_NUM
        Textfield (85,91 60x30), "%2.2f", text variable: GVL.astAxes[MAIN.hmiAxisSelection].stConfig.astMultiMasterAxis[1].fRatio
            OnMouseClick: write the text variable via Default
        Textfield (80,55 70x30), "fRatio", text list: "languageSupport", text index: "gearRatio"
        Button (12,445 168x30), "gearInMultiMaster", text list: "languageSupport", text index: "gearIn"
            OnMouseClick: execute { GVL.astAxes[Main.hmiAxisSelection].stControl.eCommand:=E_MotionFunctions.eGearInMultiMaster; GVL.astAxes[Main.hmiAxisSelection].stControl.bExecute:=TRUE; }
        SpinControl (15,181 60x30), variable: GVL.astAxes[MAIN.hmiAxisSelection].stConfig.astMultiMasterAxis[2].nIndex
            p651134158: GVL_APP.nAXIS_NUM
        SpinControl (15,271 60x30), variable: GVL.astAxes[MAIN.hmiAxisSelection].stConfig.astMultiMasterAxis[3].nIndex
            p651134158: GVL_APP.nAXIS_NUM
        SpinControl (15,361 60x30), variable: GVL.astAxes[MAIN.hmiAxisSelection].stConfig.astMultiMasterAxis[4].nIndex
            p651134158: GVL_APP.nAXIS_NUM
        Textfield (85,181 60x30), "%2.2f", text variable: GVL.astAxes[MAIN.hmiAxisSelection].stConfig.astMultiMasterAxis[2].fRatio
            OnMouseClick: write the text variable via Default
        Textfield (85,271 60x30), "%2.2f", text variable: GVL.astAxes[MAIN.hmiAxisSelection].stConfig.astMultiMasterAxis[3].fRatio
            OnMouseClick: write the text variable via Default
        Textfield (85,361 60x30), "%2.2f", text variable: GVL.astAxes[MAIN.hmiAxisSelection].stConfig.astMultiMasterAxis[4].fRatio
            OnMouseClick: write the text variable via Default
        Button (11,488 170x30), "gearOut", text list: "languageSupport", text index: "gearOut"
            OnMouseClick: execute { GVL.astAxes[Main.hmiAxisSelection].stControl.eCommand:=E_MotionFunctions.eGearOut; GVL.astAxes[Main.hmiAxisSelection].stControl.bExecute:=TRUE; }
        Textfield (9,54 70x30), "nIndex", text list: "languageSupport", text index: "masterGear"
        Textfield (85,127 60x30), "%2.2f", text variable: GVL.astAxes[MAIN.hmiAxisSelection].Axis.PlcToNc.GearRatio1
        Textfield (15,127 60x30), "%x", text variable: GVL.astAxes[MAIN.hmiAxisSelection].stConfig.astMultiMasterAxisLatched[1].nIndex
        Textfield (85,217 60x30), "%2.2f", text variable: GVL.astAxes[MAIN.hmiAxisSelection].Axis.PlcToNc.GearRatio2
        Textfield (15,217 60x30), "%x", text variable: GVL.astAxes[MAIN.hmiAxisSelection].stConfig.astMultiMasterAxisLatched[2].nIndex
        Textfield (85,307 60x30), "%2.2f", text variable: GVL.astAxes[MAIN.hmiAxisSelection].Axis.PlcToNc.GearRatio3
        Textfield (15,307 60x30), "%x", text variable: GVL.astAxes[MAIN.hmiAxisSelection].stConfig.astMultiMasterAxisLatched[3].nIndex
        Textfield (85,398 60x30), "%2.2f", text variable: GVL.astAxes[MAIN.hmiAxisSelection].Axis.PlcToNc.GearRatio4
        Textfield (15,398 60x30), "%x", text variable: GVL.astAxes[MAIN.hmiAxisSelection].stConfig.astMultiMasterAxisLatched[4].nIndex
        Lamp1 (155,399 25x25), variable: GVL.astAxes[MAIN.hmiAxisSelection].stStatus.bCoupledGear4, style: Lamp-Lamp1-Yellow
        Lamp1 (155,308 25x25), variable: GVL.astAxes[MAIN.hmiAxisSelection].stStatus.bCoupledGear3, style: Lamp-Lamp1-Yellow
        Lamp1 (155,218 25x25), variable: GVL.astAxes[MAIN.hmiAxisSelection].stStatus.bCoupledGear2, style: Lamp-Lamp1-Yellow
        Lamp1 (155,128 25x25), variable: GVL.astAxes[MAIN.hmiAxisSelection].stStatus.bCoupledGear1, style: Lamp-Lamp1-Yellow
        Lamp1 (27,7 50x50), variable: GVL.astAxes[MAIN.hmiAxisSelection].stStatus.bGeared, style: Lamp-Lamp1-Yellow
    GroupBox (10,50 190x210)
        Rectangle (0,0 190x210)
        GroupBox (3,96 73x110)
        GroupBox (92,96 86x110)
        Textfield (60,50 92x26), "ENABLE", text list: 'languageSupport', text index: "enable"
        PushSwitchLed (16,118 35x42), variable: GVL.astAxes[MAIN.hmiAxisSelection].stInputs.bLimitFwd, behaviour: TOGGLE, style: Switch-PushSwitchLed-Yellow
        PushSwitchLed (16,170 36x39), variable: GVL.astAxes[MAIN.hmiAxisSelection].stInputs.bLimitBwd, behaviour: TOGGLE, style: Switch-PushSwitchLed-Yellow
        SpinControl (108,10 72x30), variable: MAIN.hmiAxisSelection
            p651134158: GVL_APP.nAXIS_NUM
        Textfield (23,13 86x25), "axisSel", text variable: GVL_APP.nAXIS_NUM, text list: "languageSupport", text index: "axisSel"
        PowerSwitch (10,38 50x53), variable: GVL.astAxes[MAIN.hmiAxisSelection].stControl.bEnable, behaviour: TOGGLE, style: Switch-PowerSwitch-Green
        PushSwitchLed (117,118 35x42), variable: GVL.astAxes[MAIN.hmiAxisSelection].stControl.bInterlockFwd, behaviour: TOGGLE, style: Switch-PushSwitchLed-Yellow
        PushSwitchLed (117,170 36x39), variable: GVL.astAxes[MAIN.hmiAxisSelection].stControl.bInterlockBwd, behaviour: TOGGLE, style: Switch-PushSwitchLed-Yellow
        Textfield (6,94 76x26), "Fwd Enable", text list: 'languageSupport', text index: "enFW"
        Textfield (6,148 76x26), "Bwd Enable", text list: 'languageSupport', text index: "enBW"
        Textfield (96,94 76x26), "Interlock Fwd", text list: 'languageSupport', text index: "bAxisInterlockFwd"
        Textfield (96,148 76x26), "Interlock Bwd", text list: 'languageSupport', text index: "bAxisInterlockBwd"
    Textfield (10,10 231x30), "AXESMAX", text variable: GVL_APP.nAXIS_NUM, text list: "languageSupport", text index: "axesAvailable"
    Button (427,63 150x30), "moveAbsolute", text list: "languageSupport", text index: "moveAbsolute"
        OnMouseClick: execute { GVL.astAxes[MAIN.hmiAxisSelection].stControl.eCommand:=E_MotionFunctions.eMoveAbsolute; GVL.astAxes[MAIN.hmiAxisSelection].stControl.bExecute:=TRUE; }
    Button (427,143 150x30), "moveVelocity", input disabled if: GVL.astAxes[MAIN.hmiAxisSelection].stStatus.bGeared, text list: "languageSupport", text index: "moveVelocity"
        OnMouseClick: execute { GVL.astAxes[Main.hmiAxisSelection].stControl.eCommand:=E_MotionFunctions.eMoveVelocity; GVL.astAxes[Main.hmiAxisSelection].stControl.bExecute:=TRUE; }
    Button (427,103 150x30), "moveRelative", input disabled if: GVL.astAxes[MAIN.hmiAxisSelection].stStatus.bGeared, text list: "languageSupport", text index: "moveRelative"
        OnMouseClick: execute { GVL.astAxes[Main.hmiAxisSelection].stControl.eCommand:=E_MotionFunctions.eMoveRelative; GVL.astAxes[Main.hmiAxisSelection].stControl.bExecute:=TRUE; }
    Button (427,183 150x30), "moveModulo", input disabled if: GVL.astAxes[MAIN.hmiAxisSelection].stStatus.bGeared, text list: "languageSupport", text index: "moveModulo"
        OnMouseClick: execute { GVL.astAxes[Main.hmiAxisSelection].stControl.eCommand:=E_MotionFunctions.eMoveModulo; GVL.astAxes[Main.hmiAxisSelection].stControl.bExecute:=TRUE; }
    Button (587,63 150x70), "stop", pressed state: GVL.astAxes[Main.hmiAxisSelection].stControl.bStop, input disabled if: GVL.astAxes[MAIN.hmiAxisSelection].stStatus.bGeared, text list: "languageSupport", text index: "stop"
        toggle GVL.astAxes[Main.hmiAxisSelection].stControl.bStop
    Button (427,223 150x30), "jogBw", text list: "languageSupport", text index: "jogBw"
        OnMouseDown: execute {
            GVL.astAxes[Main.hmiAxisSelection].stControl.eCommand:=E_MotionFunctions.eMoveVelocity;
            GVL.astAxes[Main.hmiAxisSelection].stControl.fVelocity:=-ABS(GVL.astAxes[Main.hmiAxisSelection].stControl.fJogVelocity)
            GVL.astAxes[Main.hmiAxisSelection].stControl.bExecute:= TRUE;
        }
        OnMouseClick: execute {  }
        OnMouseUp: execute { GVL.astAxes[Main.hmiAxisSelection].stControl.bHalt:= TRUE; }
    Button (587,223 150x30), "jogFw", text list: "languageSupport", text index: "jogFw"
        OnMouseDown: execute {
            GVL.astAxes[Main.hmiAxisSelection].stControl.eCommand:=E_MotionFunctions.eMoveVelocity;
            GVL.astAxes[Main.hmiAxisSelection].stControl.fVelocity:=ABS(GVL.astAxes[Main.hmiAxisSelection].stControl.fJogVelocity)
            GVL.astAxes[Main.hmiAxisSelection].stControl.bExecute:= TRUE;
        }
        OnMouseClick: execute {  }
        OnMouseUp: execute { GVL.astAxes[Main.hmiAxisSelection].stControl.bHalt:= TRUE; }
    GroupBox (10,270 190x150)
        Rectangle (0,0 190x150)
        Textfield (90,70 90x30), "errID", text list: "languageSupport", text index: "errID"
        Textfield (10,70 80x30), "%x", text variable: GVL.astAxes[MAIN.hmiAxisSelection].stStatus.nErrorID
        Lamp1 (10,10 50x50), variable: GVL.astAxes[MAIN.hmiAxisSelection].stStatus.bError, style: Lamp-Lamp1-Red
        Textfield (60,20 120x30), "bError", text list: "languageSupport", text index: "bError"
        Button (10,110 170x30), "reset", pressed state: GVL.astAxes[Main.hmiAxisSelection].stControl.bReset, text list: "languageSupport", text index: "reset"
            OnMouseClick: toggle GVL.astAxes[Main.hmiAxisSelection].stControl.bReset
    GroupBox (10,430 190x271)
        Rectangle (0,0 190x270)
        Lamp1 (10,10 30x30), variable: GVL.astAxes[MAIN.hmiAxisSelection].stStatus.bEnabled, style: Lamp-Lamp1-Green
        Textfield (40,10 140x30), "bEnabled", text list: "languageSupport", text index: "bEnabled"
        Lamp1 (10,40 30x30), variable: GVL.astAxes[MAIN.hmiAxisSelection].stStatus.bCommandAborted, style: Lamp-Lamp1-Yellow
        Textfield (40,40 140x30), "bCommandAborted", text list: "languageSupport", text index: "bWarning"
        Textfield (40,70 140x30), "bBusy", text list: "languageSupport", text index: "bBusy"
        Lamp1 (10,100 30x30), variable: GVL.astAxes[MAIN.hmiAxisSelection].stStatus.bDone, style: Lamp-Lamp1-Green
        Textfield (40,100 140x30), "bDone", text list: 'languageSupport', text index: "bDone"
        Lamp1 (10,129 30x30), variable: GVL.astAxes[MAIN.hmiAxisSelection].stStatus.bHomed, style: Lamp-Lamp1-Green
        Textfield (40,129 140x30), "bHomed", text list: "languageSupport", text index: "bHomed"
        Lamp1 (10,159 30x30), variable: GVL.astAxes[MAIN.hmiAxisSelection].stStatus.bFwEnabled AND NOT GVL.astAxes[MAIN.hmiAxisSelection].stStatus.bInterlockedFwd, style: Lamp-Lamp1-Green
        Lamp1 (10,189 30x30), variable: GVL.astAxes[MAIN.hmiAxisSelection].stStatus.bBwEnabled AND NOT GVL.astAxes[MAIN.hmiAxisSelection].stStatus.bInterlockedBwd, style: Lamp-Lamp1-Green
        Textfield (40,159 140x30), "bFwEnabled", text list: "languageSupport", text index: "bFwEnabled"
        Textfield (40,189 140x30), "bBwEnabled", text list: "languageSupport", text index: "bBwEnabled"
        Lamp1 (9,71 30x30), variable: GVL.astAxes[MAIN.hmiAxisSelection].stStatus.bBusy, style: Lamp-Lamp1-Yellow
        Lamp1 (10,220 30x30), variable: GVL.astAxes[MAIN.hmiAxisSelection].stStatus.bInVelocity, style: Lamp-Lamp1-Green
    GroupBox (211,50 190x210)
        Rectangle (0,0 190x210)
        Textfield (10,80 100x30), "fVelocity", text list: "languageSupport", text index: "fVelocity"
        Textfield (110,80 70x30), "%2.2f", text variable: GVL.astAxes[MAIN.hmiAxisSelection].stControl.fVelocity
            OnMouseClick: write the text variable via Default
        Textfield (10,110 100x30), "fAcceleration", text list: "languageSupport", text index: "fAcceleration"
        Textfield (110,110 70x30), "%2.2f", text variable: GVL.astAxes[MAIN.hmiAxisSelection].stControl.fAcceleration
            OnMouseClick: write the text variable via Default
        Textfield (10,140 100x30), "fDeceleration", text list: "languageSupport", text index: "fDeceleration"
        Textfield (110,140 70x30), "%2.2f", text variable: GVL.astAxes[MAIN.hmiAxisSelection].stControl.fDeceleration
            OnMouseClick: write the text variable via Default
        Textfield (10,170 100x30), "fPosition", text list: "languageSupport", text index: "fPosition"
        Textfield (110,170 70x30), "%2.2f", text variable: GVL.astAxes[MAIN.hmiAxisSelection].stControl.fPosition
            OnMouseClick: write the text variable via Default
        Textfield (109,11 70x30), "%2.2f", text variable: GVL.astAxes[MAIN.hmiAxisSelection].stStatus.fActPosition
        Textfield (9,11 100x30), "actPos", text list: "languageSupport", text index: "actposition"
        Textfield (9,41 100x30), "actVel", text list: "languageSupport", text index: "actVelocity"
        Textfield (109,41 70x30), "%2.2f", text variable: GVL.astAxes[MAIN.hmiAxisSelection].stStatus.fActVelocity
    Button (428,310 150x30), "eHomeToRef_Bwd", input disabled if: GVL.astAxes[MAIN.hmiAxisSelection].stStatus.bGeared, text list: 'languageSupport', text index: "eHomeToRef_Bwd"
        OnMouseClick: execute {
            GVL.astAxes[Main.hmiAxisSelection].stControl.eCommand:=E_MotionFunctions.eHome;
            GVL.astAxes[Main.hmiAxisSelection].stConfig.eHomeSeq:=E_HomingRoutines.eHomeToRef_Bwd;
            GVL.astAxes[Main.hmiAxisSelection].stControl.bExecute:=TRUE;
        }
    Button (587,310 150x30), "eHomeToRef_Fwd", input disabled if: GVL.astAxes[MAIN.hmiAxisSelection].stStatus.bGeared, text list: "languageSupport", text index: "eHomeToRef_Fwd"
        OnMouseClick: execute {
            GVL.astAxes[Main.hmiAxisSelection].stControl.eCommand:=E_MotionFunctions.eHome;
            GVL.astAxes[Main.hmiAxisSelection].stConfig.eHomeSeq:=E_HomingRoutines.eHomeToRef_Fwd;
            GVL.astAxes[Main.hmiAxisSelection].stControl.bExecute:=TRUE;
        }
    Textfield (296,288 93x30), "bGeared", text list: "languageSupport", text index: "bGeared"
    Button (428,350 150x30), "eHomeToEncPulse_Bwd", input disabled if: GVL.astAxes[MAIN.hmiAxisSelection].stStatus.bGeared, text list: 'languageSupport', text index: "eHomeToEncPulse_Bwd"
        OnMouseClick: execute {
            GVL.astAxes[Main.hmiAxisSelection].stControl.eCommand:=E_MotionFunctions.eHome;
            GVL.astAxes[Main.hmiAxisSelection].stConfig.eHomeSeq:=E_HomingRoutines.eHomeToEncPulse_Bwd;
            GVL.astAxes[Main.hmiAxisSelection].stControl.bExecute:=TRUE;
        }
    Button (587,350 150x30), "eHomeToEncPulse_Fwd", input disabled if: GVL.astAxes[MAIN.hmiAxisSelection].stStatus.bGeared, text list: "languageSupport", text index: "eHomeToEncPulse_Fwd"
        OnMouseClick: execute {
            GVL.astAxes[Main.hmiAxisSelection].stControl.eCommand:=E_MotionFunctions.eHome;
            GVL.astAxes[Main.hmiAxisSelection].stConfig.eHomeSeq:=E_HomingRoutines.eHomeToEncPulse_Fwd;
            GVL.astAxes[Main.hmiAxisSelection].stControl.bExecute:=TRUE;
        }
    Button (428,470 150x30), "eHomeDirect", input disabled if: GVL.astAxes[MAIN.hmiAxisSelection].stStatus.bGeared, text list: 'languageSupport', text index: "eHomeDirect"
        OnMouseClick: execute {
            GVL.astAxes[Main.hmiAxisSelection].stControl.eCommand:=E_MotionFunctions.eHome;
            GVL.astAxes[Main.hmiAxisSelection].stConfig.eHomeSeq:=E_HomingRoutines.eHomeDirect;
            GVL.astAxes[Main.hmiAxisSelection].stControl.bExecute:=TRUE;
        }
    Button (428,270 150x30), "eHomeToLimit_Bwd", input disabled if: GVL.astAxes[MAIN.hmiAxisSelection].stStatus.bGeared, text list: 'languageSupport', text index: "eHomeToLimit_Bwd"
        OnMouseClick: execute {
            GVL.astAxes[Main.hmiAxisSelection].stControl.eCommand:=E_MotionFunctions.eHome;
            GVL.astAxes[Main.hmiAxisSelection].stConfig.eHomeSeq:=E_HomingRoutines.eHomeToLimit_Bwd;
            GVL.astAxes[Main.hmiAxisSelection].stControl.bExecute:=TRUE;
        }
    Button (587,270 150x30), "eHomeToLimit_Fwd", input disabled if: GVL.astAxes[MAIN.hmiAxisSelection].stStatus.bGeared, text list: "languageSupport", text index: "eHomeToLimit_Fwd"
        OnMouseClick: execute {
            GVL.astAxes[Main.hmiAxisSelection].stControl.eCommand:=E_MotionFunctions.eHome;
            GVL.astAxes[Main.hmiAxisSelection].stConfig.eHomeSeq:=E_HomingRoutines.eHomeToLimit_Fwd;
            GVL.astAxes[Main.hmiAxisSelection].stControl.bExecute:=TRUE;
        }
    Textfield (428,540 150x30), "%2.2f", text variable: GVL.astAxes[MAIN.hmiAxisSelection].stConfig.fHomePosition
        OnMouseClick: write the text variable via Default
    Button (428,390 150x30), "eHomeToEncPulse_viaBwdLimit", input disabled if: GVL.astAxes[MAIN.hmiAxisSelection].stStatus.bGeared, text list: 'languageSupport', text index: "eHomeToEncPulse_viaBwdLimit"
        OnMouseClick: execute {
            GVL.astAxes[Main.hmiAxisSelection].stControl.eCommand:=E_MotionFunctions.eHome;
            GVL.astAxes[Main.hmiAxisSelection].stConfig.eHomeSeq:=E_HomingRoutines.eHomeToEncPulse_viaBwdLimit;
            GVL.astAxes[Main.hmiAxisSelection].stControl.bExecute:=TRUE;
        }
    Button (587,390 150x30), "eHomeToEncPulse_viaFwdLimit", input disabled if: GVL.astAxes[MAIN.hmiAxisSelection].stStatus.bGeared, text list: "languageSupport", text index: "eHomeToEncPulse_viaFwdLimit"
        OnMouseClick: execute {
            GVL.astAxes[Main.hmiAxisSelection].stControl.eCommand:=E_MotionFunctions.eHome;
            GVL.astAxes[Main.hmiAxisSelection].stConfig.eHomeSeq:=E_HomingRoutines.eHomeToEncPulse_viaFwdLimit;
            GVL.astAxes[Main.hmiAxisSelection].stControl.bExecute:=TRUE;
        }
    Textfield (588,540 150x30), "%2.2f", text variable: GVL.astAxes[MAIN.hmiAxisSelection].stConfig.fHomeFinishDistance
        OnMouseClick: write the text variable via Default
    Textfield (428,510 150x30), "fHomePosition", text list: "languageSupport", text index: "fHomePosition"
    Textfield (588,510 150x30), "fHomeFinishDistance", text list: "languageSupport", text index: "fHomeFinishDistance"
    Group (602,14 150x30)
        Button (0,0 150x30), "bLocalMode", text list: 'languageSupport', text index: bLocalMode
            OnMouseClick: toggle bLocalMode
        Lamp1 (5,3 25x25), variable: bLocalMode, style: Lamp-Lamp1-Green
    Rectangle (763,50 192x307)
    Button (780,146 157x30), "eWriteParameter", input disabled if: GVL.astAxes[MAIN.hmiAxisSelection].stStatus.bGeared, text list: "languageSupport", text index: "eWriteParameter"
        OnMouseClick: execute { GVL.astAxes[MAIN.hmiAxisSelection].stControl.eCommand:=E_MotionFunctions.eWriteParameter; GVL.astAxes[MAIN.hmiAxisSelection].stControl.bExecute:=TRUE; }
    Textfield (772,62 170x30), "%x", text variable: astAxes[MAIN.hmiAxisSelection].stConfig.eAxisParameters
        OnMouseClick: write GVL.astAxes[MAIN.hmiAxisSelection].stConfig.eAxisParameters via Default
    Textfield (762,107 120x30), "fWriteAxisParameter", text list: "languageSupport", text index: "fWriteAxisParameter"
    Textfield (882,107 60x30), "%2.4f", text variable: astAxes[MAIN.hmiAxisSelection].stConfig.fWriteAxisParameter
        OnMouseClick: write GVL.astAxes[MAIN.hmiAxisSelection].stConfig.fWriteAxisParameter via Default
    Textfield (886,266 60x30), "%2.4f", text variable: astAxes[MAIN.hmiAxisSelection].stConfig.fReadAxisParameter
        OnMouseClick: write GVL.astAxes[MAIN.hmiAxisSelection].stConfig.fReadAxisParameter via Default
    Textfield (766,266 120x30), "fReadAxisParameter", text list: "languageSupport", text index: "fReadAxisParameter"
    Button (781,209 156x31), "eReadParameter", input disabled if: GVL.astAxes[MAIN.hmiAxisSelection].stStatus.bGeared, text list: 'languageSupport', text index: "eReadParameter"
        OnMouseClick: execute { GVL.astAxes[MAIN.hmiAxisSelection].stControl.eCommand:=E_MotionFunctions.eReadParameter; GVL.astAxes[MAIN.hmiAxisSelection].stControl.bExecute:=TRUE; }
    ComboBoxInteger (767,12 304x30), variable: GVL.astAxes[MAIN.hmiAxisSelection].stConfig.eAxisParameters, text list: 'ParameterTextList'
    Textfield (50,650 140x30), "bInVelocity", text list: 'languageSupport', text index: "bInVelocity"
    Button (587,430 150x30), "eHomeToBlock_Fwd", input disabled if: GVL.astAxes[MAIN.hmiAxisSelection].stStatus.bGeared, text list: "languageSupport", text index: "eHomeToBlock_Fwd"
        OnMouseClick: execute {
            GVL.astAxes[Main.hmiAxisSelection].stControl.eCommand:=E_MotionFunctions.eHome;
            GVL.astAxes[Main.hmiAxisSelection].stConfig.eHomeSeq:=E_HomingRoutines.eHomeToBlock_Fwd;
            GVL.astAxes[Main.hmiAxisSelection].stControl.bExecute:=TRUE;
        }
END_VISUALIZATION
